// TIA Portal V20 export
FUNCTION_BLOCK "Sequence_1_ManualInput"   // FB126, LAD
TITLE = Sequence
// Sequence template programmend in ladder logic
// stored: IsIECCheckEnabled true, MemoryReserve 100, Namespace Unit1.Em5, SetENOAutomatically true
   VAR
      statSelectedJobNumber { ExternalWritable := 'False'} : DInt;   // Evaluated Job Number
      instSequenceLADControl { ExternalWritable := 'False'} : "LAF_ControlLadSequence";
      instSequenceLADStatus { ExternalWritable := 'False'} : "LAF_StatusLadSequence";
      statAxisCmdNumber { ExternalWritable := 'False'} : Array[0..1] of USInt;
      statTwoWayActCmdNumber { ExternalWritable := 'False'} : Array[0..3] of USInt;
      statPulse { ExternalWritable := 'False'} : Array[0..999] of Bool;
      statTonTimer { ExternalWritable := 'False'} : Array[0..999] of TON_TIME;
   END_VAR
   VAR_TEMP
      tempCustomerAction : Bool;   // Placeholder for possible actions
      tempDo_nothing_and_wait_for_init : Bool;   // Placeholder for doing nothing
      tempSafeStateCondition : Bool;   // Temp Condition for the equipment module to be in a safe state
   END_VAR
   VAR CONSTANT
      STEP_IDLE : DInt := 1;   // Idle Step
      JOB_1_STEP_01 : DInt := 101;   // Template Step
      JOB_1_STEP_11 : DInt := 111;   // Template Step
      JOB_1_STEP_21 : DInt := 121;   // Template Step
      JOB_1_STEP_31 : DInt := 131;   // Template Step
      JOB_1_STEP_41 : DInt := 141;
      JOB_1_STEP_51 : DInt := 151;
      JOB_1_STEP_91 : DInt := 191;
      JOB_2_STEP_01 : DInt := 201;   // Template Step
      JOB_2_STEP_11 : DInt := 211;   // Template Step
      JOB_2_STEP_21 : DInt := 221;   // Template Step
      JOB_2_STEP_31 : DInt := 231;   // Template Step
      JOB_2_STEP_41 : DInt := 241;   // Template Step
      JOB_2_STEP_51 : DInt := 251;   // Template Step
      JOB_2_STEP_61 : DInt := 261;   // Template Step
      JOB_2_STEP_91 : DInt := 291;   // Template Step
      JOB_3_STEP_01 : DInt := 301;   // Template Step
      JOB_3_STEP_11 : DInt := 311;   // Template Step
      JOB_3_STEP_21 : DInt := 321;   // Template Step
      JOB_3_STEP_31 : DInt := 331;   // Template Step
      JOB_3_STEP_41 : DInt := 341;   // Template Step
      JOB_3_STEP_51 : DInt := 351;   // Template Step
      JOB_3_STEP_91 : DInt := 391;   // Template Step
      STEP_IMMEDIATE_STOP : DInt := 901;   // Step executed when an immediate stop command is triggered for the sequence (i.e. when unit is in state aborting)
      SeqDelayTime : Time := T#100ms;
      SeqNoDelayTime : Time := T#0ms;
      TRUE : Bool := TRUE;
      FALSE : Bool := FALSE;
      NgAndManualInputAxisYHomePos : SInt := 0;
      NgAndManualInputAxisYWorkPos : SInt := 1;
   END_VAR
   // // statAxisCmdNumber[0] : cmNgAndManualInputAxisY
   // // statAxisCmdNumber[1] : cmMagazineAxisZ
   // // statTwoWayActCmdNumber[0] : cmNgAndManualInputCylinderUpDown
   // // statTwoWayActCmdNumber[1] : cmNgAndManualInputVacuum1OnOff
   // // statTwoWayActCmdNumber[2] : cmNgAndManualInputVacuum2OnOff
   // // statTwoWayActCmdNumber[3] : cmMagazineLockCylinderUpDown
   VAR_TEMP   // added for the SCL form of the ladder/FBD networks
      _w1 : Bool;
      _w2 : Bool;
      _w3 : Bool;
   END_VAR
BEGIN

REGION Network 1: BLOCK INFO HEADER
   // (company) / (C) Copyright (year)
   // ---------------------------------------------------------------------------------
   // Title:                             (Title of this block)
   // Comment/Function: (that is implemented in the block)
   // Library/Family:           (that the source is dedicated to)
   // Author:                        (department / person in charge / contact)
   // Target System:          (test system with FW version)
   // Engineering:              TIA Portal (SW version)
   // Restrictions:               (OB types, etc.)
   // Requirements:           (hardware, technological package, etc.)
   // ---------------------------------------------------------------------------------
   // Change log table:
   // Version          | Date             | Signature      | Expert in charge  | Changes applied ------------------------|----------------------|-------------------------|--------------------------------|-----------------------
   // 001.000.000 | yyyy-mm-dd | 0x00000000 | (name of expert) | First released version
END_REGION

REGION Network 2: DESCRIPTION
   // This is a template block provided by the Automation Framework. It can be used to create an own project.
   // The Block Info Header is prepared to put in your own data.
   // Description of the block could be added here and the docu created by Code2Docu.
END_REGION

REGION Network 3: ******************** CONTROL ********************
END_REGION

REGION Network 4: Sequence Control
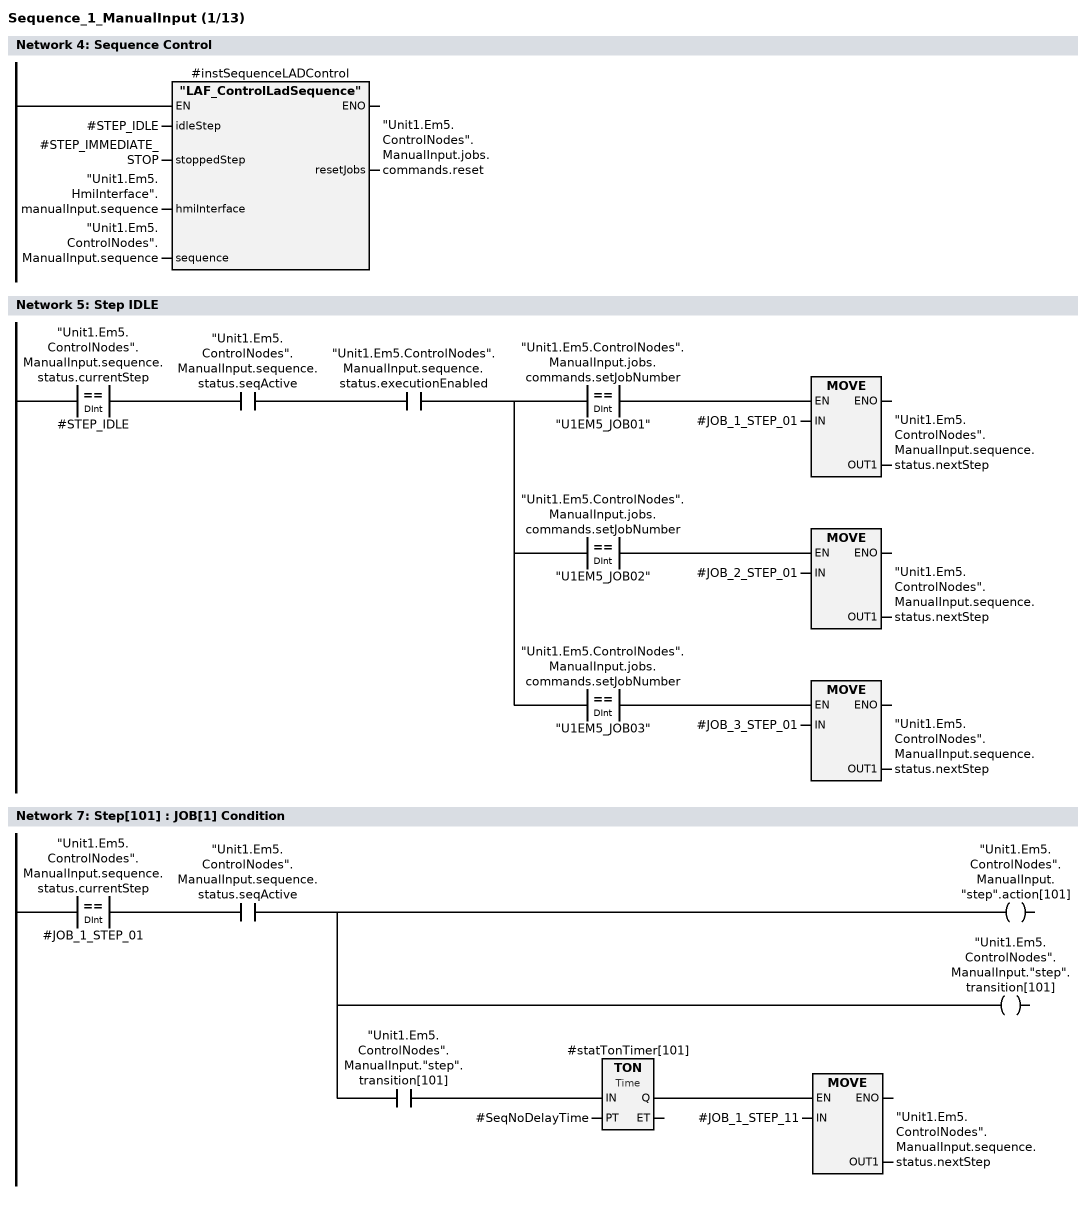
   RUNG wire#powerrail
      #instSequenceLADControl(idleStep := #STEP_IDLE, stoppedStep := #STEP_IMMEDIATE_STOP, hmiInterface := "Unit1.Em5.HmiInterface".manualInput.sequence, sequence := "Unit1.Em5.ControlNodes".ManualInput.sequence, resetJobs => "Unit1.Em5.ControlNodes".ManualInput.jobs.commands.reset)
   END_RUNG
   // the same network as SCL:
   #instSequenceLADControl(idleStep := #STEP_IDLE,   // "LAF_ControlLadSequence"
                           stoppedStep := #STEP_IMMEDIATE_STOP,
                           hmiInterface := "Unit1.Em5.HmiInterface".manualInput.sequence,
                           sequence := "Unit1.Em5.ControlNodes".ManualInput.sequence,
                           resetJobs => "Unit1.Em5.ControlNodes".ManualInput.jobs.commands.reset);
END_REGION

REGION Network 5: Step IDLE
   RUNG wire#powerrail
      { S7_Templates := "SrcType := DInt" } EQ_Contact(in1 := "Unit1.Em5.ControlNodes".ManualInput.sequence.status.currentStep, in2 := #STEP_IDLE)
      Contact( "Unit1.Em5.ControlNodes".ManualInput.sequence.status.seqActive )
      Contact( "Unit1.Em5.ControlNodes".ManualInput.sequence.status.executionEnabled )
      wire#w1
      { S7_Templates := "SrcType := DInt" } EQ_Contact(in1 := "Unit1.Em5.ControlNodes".ManualInput.jobs.commands.setJobNumber, in2 := "U1EM5_JOB01")
      Move(in := #JOB_1_STEP_01, out1 => "Unit1.Em5.ControlNodes".ManualInput.sequence.status.nextStep)
   END_RUNG
   RUNG wire#w1
      { S7_Templates := "SrcType := DInt" } EQ_Contact(in1 := "Unit1.Em5.ControlNodes".ManualInput.jobs.commands.setJobNumber, in2 := "U1EM5_JOB02")
      Move(in := #JOB_2_STEP_01, out1 => "Unit1.Em5.ControlNodes".ManualInput.sequence.status.nextStep)
   END_RUNG
   RUNG wire#w1
      { S7_Templates := "SrcType := DInt" } EQ_Contact(in1 := "Unit1.Em5.ControlNodes".ManualInput.jobs.commands.setJobNumber, in2 := "U1EM5_JOB03")
      Move(in := #JOB_3_STEP_01, out1 => "Unit1.Em5.ControlNodes".ManualInput.sequence.status.nextStep)
   END_RUNG
   // the same network as SCL:
   #_w1 := ("Unit1.Em5.ControlNodes".ManualInput.sequence.status.currentStep = #STEP_IDLE) AND "Unit1.Em5.ControlNodes".ManualInput.sequence.status.seqActive AND "Unit1.Em5.ControlNodes".ManualInput.sequence.status.executionEnabled;
   IF #_w1 AND ("Unit1.Em5.ControlNodes".ManualInput.jobs.commands.setJobNumber = "U1EM5_JOB01") THEN
       "Unit1.Em5.ControlNodes".ManualInput.sequence.status.nextStep := #JOB_1_STEP_01;
   END_IF;
   IF #_w1 AND ("Unit1.Em5.ControlNodes".ManualInput.jobs.commands.setJobNumber = "U1EM5_JOB02") THEN
       "Unit1.Em5.ControlNodes".ManualInput.sequence.status.nextStep := #JOB_2_STEP_01;
   END_IF;
   IF #_w1 AND ("Unit1.Em5.ControlNodes".ManualInput.jobs.commands.setJobNumber = "U1EM5_JOB03") THEN
       "Unit1.Em5.ControlNodes".ManualInput.sequence.status.nextStep := #JOB_3_STEP_01;
   END_IF;
END_REGION

REGION Network 6: ******************** JOB[1] EM INITIALIZED ********************
END_REGION

REGION Network 7: Step[101] : JOB[1] Condition
   RUNG wire#powerrail
      { S7_Templates := "SrcType := DInt" } EQ_Contact(in1 := "Unit1.Em5.ControlNodes".ManualInput.sequence.status.currentStep, in2 := #JOB_1_STEP_01)
      Contact( "Unit1.Em5.ControlNodes".ManualInput.sequence.status.seqActive )
      wire#w1
      Coil( "Unit1.Em5.ControlNodes".ManualInput."step".action[101] )
   END_RUNG
   RUNG wire#w1
      Coil( "Unit1.Em5.ControlNodes".ManualInput."step".transition[101] )
   END_RUNG
   RUNG wire#w1
      Contact( "Unit1.Em5.ControlNodes".ManualInput."step".transition[101] )
      { S7_Templates := "time_type := Time" } #statTonTimer[101].TON(pt := #SeqNoDelayTime, et =>)
      Move(in := #JOB_1_STEP_11, out1 => "Unit1.Em5.ControlNodes".ManualInput.sequence.status.nextStep)
   END_RUNG
   // the same network as SCL:
   "Unit1.Em5.ControlNodes".ManualInput."step".action[101] := ("Unit1.Em5.ControlNodes".ManualInput.sequence.status.currentStep = #JOB_1_STEP_01) AND "Unit1.Em5.ControlNodes".ManualInput.sequence.status.seqActive;
   "Unit1.Em5.ControlNodes".ManualInput."step".transition[101] := ("Unit1.Em5.ControlNodes".ManualInput.sequence.status.currentStep = #JOB_1_STEP_01) AND "Unit1.Em5.ControlNodes".ManualInput.sequence.status.seqActive;
   #statTonTimer[101].TON(IN := ("Unit1.Em5.ControlNodes".ManualInput.sequence.status.currentStep = #JOB_1_STEP_01) AND "Unit1.Em5.ControlNodes".ManualInput.sequence.status.seqActive AND "Unit1.Em5.ControlNodes".ManualInput."step".transition[101],
                          PT := #SeqNoDelayTime);
   IF #statTonTimer[101].Q THEN
       "Unit1.Em5.ControlNodes".ManualInput.sequence.status.nextStep := #JOB_1_STEP_11;
   END_IF;
END_REGION

REGION Network 8: Step[111] : Ng And Manual Input Cylinder HomePos & Magazine Lock Cylinder WorkPos Check
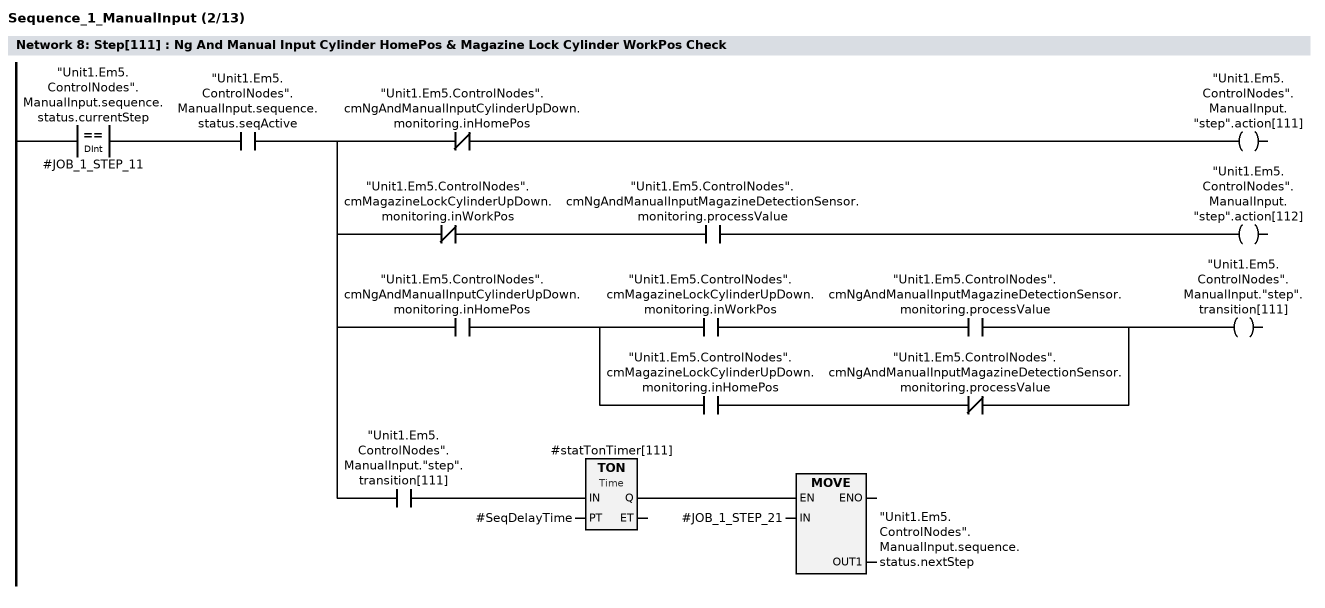
   RUNG wire#powerrail
      { S7_Templates := "SrcType := DInt" } EQ_Contact(in1 := "Unit1.Em5.ControlNodes".ManualInput.sequence.status.currentStep, in2 := #JOB_1_STEP_11)
      Contact( "Unit1.Em5.ControlNodes".ManualInput.sequence.status.seqActive )
      wire#w1
      I_Contact( "Unit1.Em5.ControlNodes".cmNgAndManualInputCylinderUpDown.monitoring.inHomePos )
      Coil( "Unit1.Em5.ControlNodes".ManualInput."step".action[111] )
   END_RUNG
   RUNG wire#w1
      I_Contact( "Unit1.Em5.ControlNodes".cmMagazineLockCylinderUpDown.monitoring.inWorkPos )
      Contact( "Unit1.Em5.ControlNodes".cmNgAndManualInputMagazineDetectionSensor.monitoring.processValue )
      Coil( "Unit1.Em5.ControlNodes".ManualInput."step".action[112] )
   END_RUNG
   RUNG wire#w1
      Contact( "Unit1.Em5.ControlNodes".cmNgAndManualInputCylinderUpDown.monitoring.inHomePos )
      wire#w2
      Contact( "Unit1.Em5.ControlNodes".cmMagazineLockCylinderUpDown.monitoring.inWorkPos )
      Contact( "Unit1.Em5.ControlNodes".cmNgAndManualInputMagazineDetectionSensor.monitoring.processValue )
      wire#w3
      Coil( "Unit1.Em5.ControlNodes".ManualInput."step".transition[111] )
   END_RUNG
   RUNG wire#w2
      Contact( "Unit1.Em5.ControlNodes".cmMagazineLockCylinderUpDown.monitoring.inHomePos )
      I_Contact( "Unit1.Em5.ControlNodes".cmNgAndManualInputMagazineDetectionSensor.monitoring.processValue )
   END_RUNG wire#w3
   RUNG wire#w1
      Contact( "Unit1.Em5.ControlNodes".ManualInput."step".transition[111] )
      { S7_Templates := "time_type := Time" } #statTonTimer[111].TON(pt := #SeqDelayTime, et =>)
      Move(in := #JOB_1_STEP_21, out1 => "Unit1.Em5.ControlNodes".ManualInput.sequence.status.nextStep)
   END_RUNG
   // the same network as SCL:
   #_w1 := ("Unit1.Em5.ControlNodes".ManualInput.sequence.status.currentStep = #JOB_1_STEP_11) AND "Unit1.Em5.ControlNodes".ManualInput.sequence.status.seqActive;
   "Unit1.Em5.ControlNodes".ManualInput."step".action[111] := #_w1 AND NOT "Unit1.Em5.ControlNodes".cmNgAndManualInputCylinderUpDown.monitoring.inHomePos;
   "Unit1.Em5.ControlNodes".ManualInput."step".action[112] := #_w1 AND NOT "Unit1.Em5.ControlNodes".cmMagazineLockCylinderUpDown.monitoring.inWorkPos AND "Unit1.Em5.ControlNodes".cmNgAndManualInputMagazineDetectionSensor.monitoring.processValue;
   "Unit1.Em5.ControlNodes".ManualInput."step".transition[111] := #_w1 AND "Unit1.Em5.ControlNodes".cmNgAndManualInputCylinderUpDown.monitoring.inHomePos AND (("Unit1.Em5.ControlNodes".cmMagazineLockCylinderUpDown.monitoring.inWorkPos AND "Unit1.Em5.ControlNodes".cmNgAndManualInputMagazineDetectionSensor.monitoring.processValue) OR ("Unit1.Em5.ControlNodes".cmMagazineLockCylinderUpDown.monitoring.inHomePos AND NOT "Unit1.Em5.ControlNodes".cmNgAndManualInputMagazineDetectionSensor.monitoring.processValue));
   #statTonTimer[111].TON(IN := #_w1 AND "Unit1.Em5.ControlNodes".ManualInput."step".transition[111],
                          PT := #SeqDelayTime);
   IF #statTonTimer[111].Q THEN
       "Unit1.Em5.ControlNodes".ManualInput.sequence.status.nextStep := #JOB_1_STEP_21;
   END_IF;
END_REGION

REGION Network 9: Step[121] : Ng And Manual Input Vacuum HomePos & Vibrator Home Pos Check
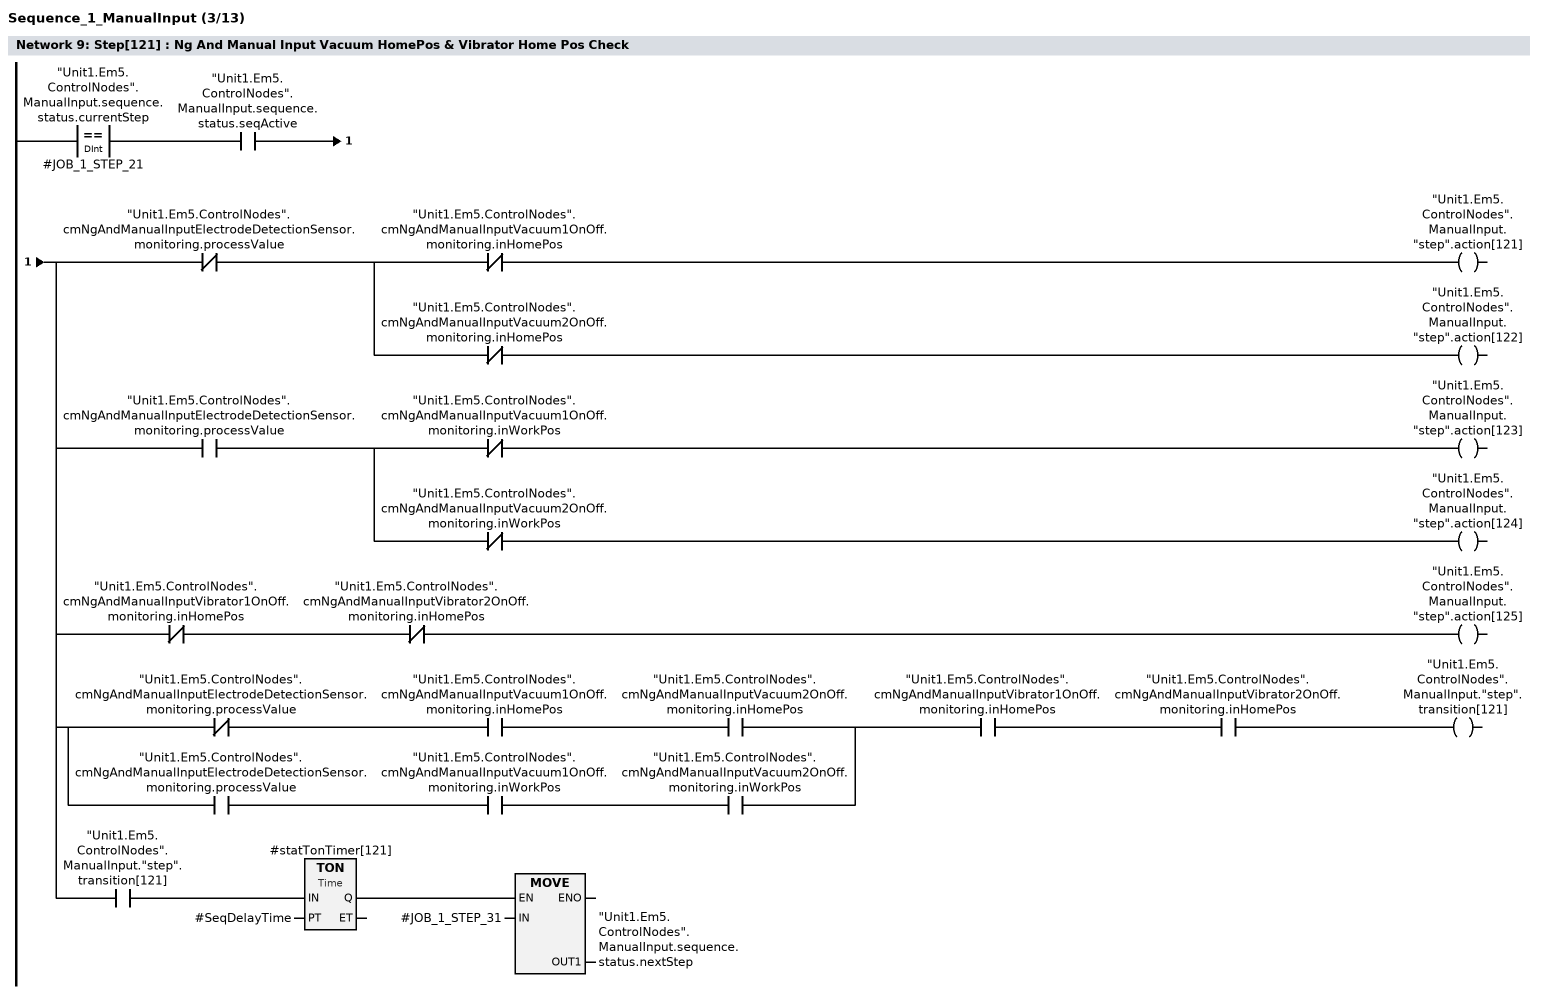
   RUNG wire#powerrail
      { S7_Templates := "SrcType := DInt" } EQ_Contact(in1 := "Unit1.Em5.ControlNodes".ManualInput.sequence.status.currentStep, in2 := #JOB_1_STEP_21)
      Contact( "Unit1.Em5.ControlNodes".ManualInput.sequence.status.seqActive )
      wire#w1
      I_Contact( "Unit1.Em5.ControlNodes".cmNgAndManualInputElectrodeDetectionSensor.monitoring.processValue )
      wire#w2
      I_Contact( "Unit1.Em5.ControlNodes".cmNgAndManualInputVacuum1OnOff.monitoring.inHomePos )
      Coil( "Unit1.Em5.ControlNodes".ManualInput."step".action[121] )
   END_RUNG
   RUNG wire#w2
      I_Contact( "Unit1.Em5.ControlNodes".cmNgAndManualInputVacuum2OnOff.monitoring.inHomePos )
      Coil( "Unit1.Em5.ControlNodes".ManualInput."step".action[122] )
   END_RUNG
   RUNG wire#w1
      Contact( "Unit1.Em5.ControlNodes".cmNgAndManualInputElectrodeDetectionSensor.monitoring.processValue )
      wire#w3
      I_Contact( "Unit1.Em5.ControlNodes".cmNgAndManualInputVacuum1OnOff.monitoring.inWorkPos )
      Coil( "Unit1.Em5.ControlNodes".ManualInput."step".action[123] )
   END_RUNG
   RUNG wire#w3
      I_Contact( "Unit1.Em5.ControlNodes".cmNgAndManualInputVacuum2OnOff.monitoring.inWorkPos )
      Coil( "Unit1.Em5.ControlNodes".ManualInput."step".action[124] )
   END_RUNG
   RUNG wire#w1
      I_Contact( "Unit1.Em5.ControlNodes".cmNgAndManualInputVibrator1OnOff.monitoring.inHomePos )
      I_Contact( "Unit1.Em5.ControlNodes".cmNgAndManualInputVibrator2OnOff.monitoring.inHomePos )
      Coil( "Unit1.Em5.ControlNodes".ManualInput."step".action[125] )
   END_RUNG
   RUNG wire#w1
      I_Contact( "Unit1.Em5.ControlNodes".cmNgAndManualInputElectrodeDetectionSensor.monitoring.processValue )
      Contact( "Unit1.Em5.ControlNodes".cmNgAndManualInputVacuum1OnOff.monitoring.inHomePos )
      Contact( "Unit1.Em5.ControlNodes".cmNgAndManualInputVacuum2OnOff.monitoring.inHomePos )
      wire#w4
      Contact( "Unit1.Em5.ControlNodes".cmNgAndManualInputVibrator1OnOff.monitoring.inHomePos )
      Contact( "Unit1.Em5.ControlNodes".cmNgAndManualInputVibrator2OnOff.monitoring.inHomePos )
      Coil( "Unit1.Em5.ControlNodes".ManualInput."step".transition[121] )
   END_RUNG
   RUNG wire#w1
      Contact( "Unit1.Em5.ControlNodes".cmNgAndManualInputElectrodeDetectionSensor.monitoring.processValue )
      Contact( "Unit1.Em5.ControlNodes".cmNgAndManualInputVacuum1OnOff.monitoring.inWorkPos )
      Contact( "Unit1.Em5.ControlNodes".cmNgAndManualInputVacuum2OnOff.monitoring.inWorkPos )
   END_RUNG wire#w4
   RUNG wire#w1
      Contact( "Unit1.Em5.ControlNodes".ManualInput."step".transition[121] )
      { S7_Templates := "time_type := Time" } #statTonTimer[121].TON(pt := #SeqDelayTime, et =>)
      Move(in := #JOB_1_STEP_31, out1 => "Unit1.Em5.ControlNodes".ManualInput.sequence.status.nextStep)
   END_RUNG
   // the same network as SCL:
   #_w1 := ("Unit1.Em5.ControlNodes".ManualInput.sequence.status.currentStep = #JOB_1_STEP_21) AND "Unit1.Em5.ControlNodes".ManualInput.sequence.status.seqActive;
   #_w2 := #_w1 AND NOT "Unit1.Em5.ControlNodes".cmNgAndManualInputElectrodeDetectionSensor.monitoring.processValue;
   "Unit1.Em5.ControlNodes".ManualInput."step".action[121] := #_w2 AND NOT "Unit1.Em5.ControlNodes".cmNgAndManualInputVacuum1OnOff.monitoring.inHomePos;
   "Unit1.Em5.ControlNodes".ManualInput."step".action[122] := #_w2 AND NOT "Unit1.Em5.ControlNodes".cmNgAndManualInputVacuum2OnOff.monitoring.inHomePos;
   #_w3 := #_w1 AND "Unit1.Em5.ControlNodes".cmNgAndManualInputElectrodeDetectionSensor.monitoring.processValue;
   "Unit1.Em5.ControlNodes".ManualInput."step".action[123] := #_w3 AND NOT "Unit1.Em5.ControlNodes".cmNgAndManualInputVacuum1OnOff.monitoring.inWorkPos;
   "Unit1.Em5.ControlNodes".ManualInput."step".action[124] := #_w3 AND NOT "Unit1.Em5.ControlNodes".cmNgAndManualInputVacuum2OnOff.monitoring.inWorkPos;
   "Unit1.Em5.ControlNodes".ManualInput."step".action[125] := #_w1 AND NOT "Unit1.Em5.ControlNodes".cmNgAndManualInputVibrator1OnOff.monitoring.inHomePos AND NOT "Unit1.Em5.ControlNodes".cmNgAndManualInputVibrator2OnOff.monitoring.inHomePos;
   "Unit1.Em5.ControlNodes".ManualInput."step".transition[121] := #_w1 AND ((NOT "Unit1.Em5.ControlNodes".cmNgAndManualInputElectrodeDetectionSensor.monitoring.processValue AND "Unit1.Em5.ControlNodes".cmNgAndManualInputVacuum1OnOff.monitoring.inHomePos AND "Unit1.Em5.ControlNodes".cmNgAndManualInputVacuum2OnOff.monitoring.inHomePos) OR ("Unit1.Em5.ControlNodes".cmNgAndManualInputElectrodeDetectionSensor.monitoring.processValue AND "Unit1.Em5.ControlNodes".cmNgAndManualInputVacuum1OnOff.monitoring.inWorkPos AND "Unit1.Em5.ControlNodes".cmNgAndManualInputVacuum2OnOff.monitoring.inWorkPos)) AND "Unit1.Em5.ControlNodes".cmNgAndManualInputVibrator1OnOff.monitoring.inHomePos AND "Unit1.Em5.ControlNodes".cmNgAndManualInputVibrator2OnOff.monitoring.inHomePos;
   #statTonTimer[121].TON(IN := #_w1 AND "Unit1.Em5.ControlNodes".ManualInput."step".transition[121],
                          PT := #SeqDelayTime);
   IF #statTonTimer[121].Q THEN
       "Unit1.Em5.ControlNodes".ManualInput.sequence.status.nextStep := #JOB_1_STEP_31;
   END_IF;
END_REGION

REGION Network 10: Step[131] : Ng And Manual Input AxisY & Magazine AxisZ Homed Check
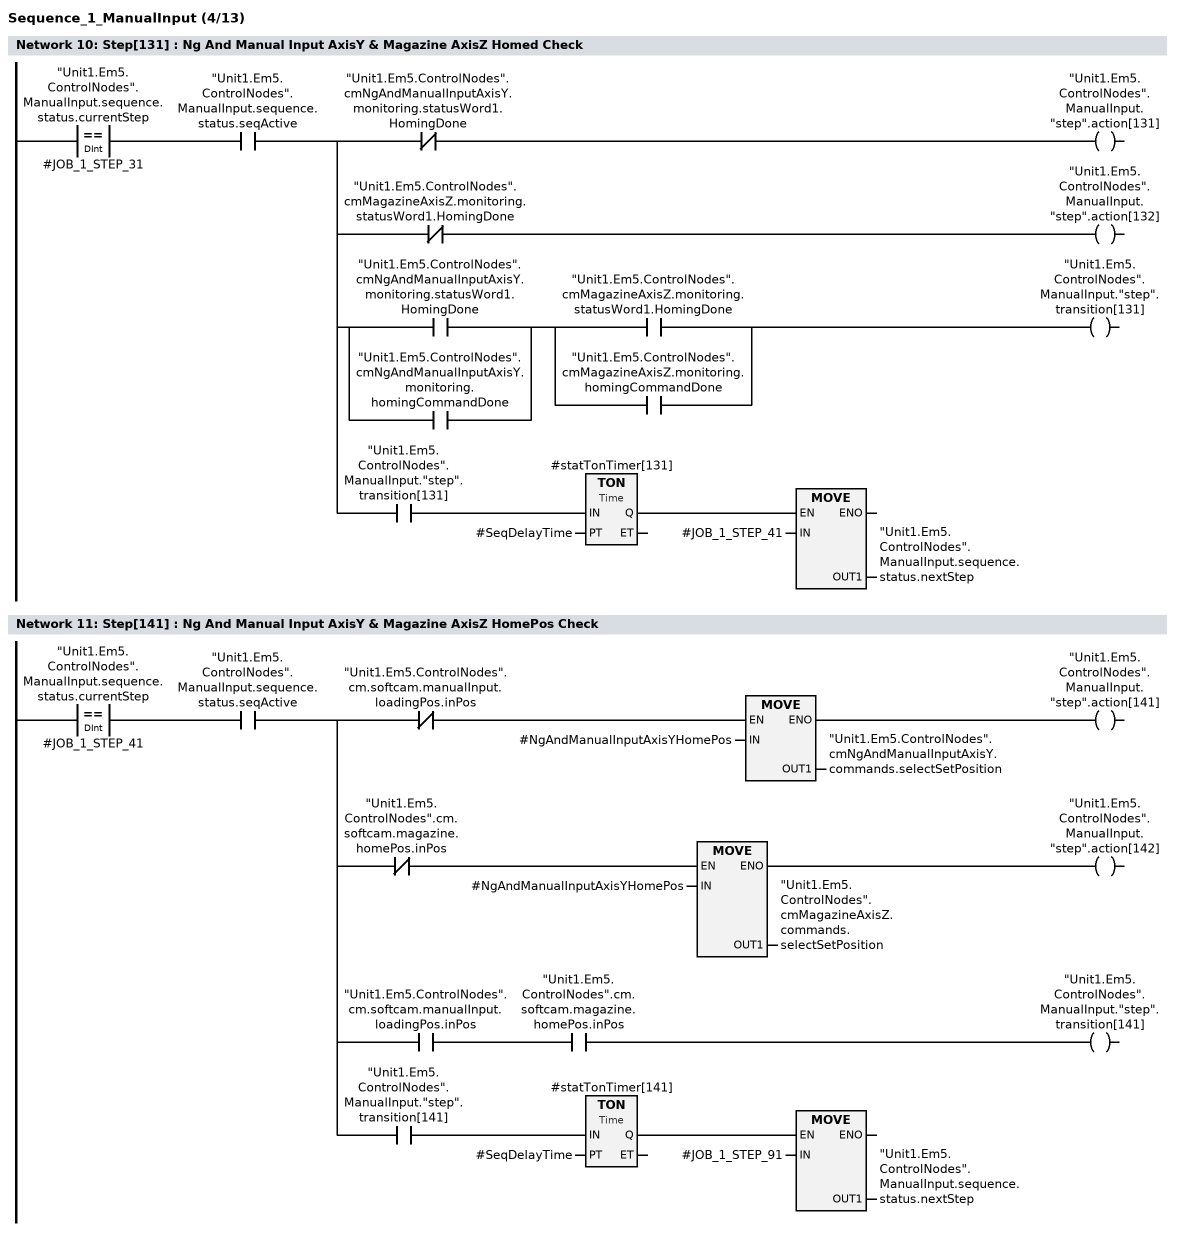
   RUNG wire#powerrail
      { S7_Templates := "SrcType := DInt" } EQ_Contact(in1 := "Unit1.Em5.ControlNodes".ManualInput.sequence.status.currentStep, in2 := #JOB_1_STEP_31)
      Contact( "Unit1.Em5.ControlNodes".ManualInput.sequence.status.seqActive )
      wire#w1
      I_Contact( "Unit1.Em5.ControlNodes".cmNgAndManualInputAxisY.monitoring.statusWord1.HomingDone )
      Coil( "Unit1.Em5.ControlNodes".ManualInput."step".action[131] )
   END_RUNG
   RUNG wire#w1
      I_Contact( "Unit1.Em5.ControlNodes".cmMagazineAxisZ.monitoring.statusWord1.HomingDone )
      Coil( "Unit1.Em5.ControlNodes".ManualInput."step".action[132] )
   END_RUNG
   RUNG wire#w1
      Contact( "Unit1.Em5.ControlNodes".cmNgAndManualInputAxisY.monitoring.statusWord1.HomingDone )
      wire#w2
      Contact( "Unit1.Em5.ControlNodes".cmMagazineAxisZ.monitoring.statusWord1.HomingDone )
      wire#w3
      Coil( "Unit1.Em5.ControlNodes".ManualInput."step".transition[131] )
   END_RUNG
   RUNG wire#w1
      Contact( "Unit1.Em5.ControlNodes".cmNgAndManualInputAxisY.monitoring.homingCommandDone )
   END_RUNG wire#w2
   RUNG wire#w2
      Contact( "Unit1.Em5.ControlNodes".cmMagazineAxisZ.monitoring.homingCommandDone )
   END_RUNG wire#w3
   RUNG wire#w1
      Contact( "Unit1.Em5.ControlNodes".ManualInput."step".transition[131] )
      { S7_Templates := "time_type := Time" } #statTonTimer[131].TON(pt := #SeqDelayTime, et =>)
      Move(in := #JOB_1_STEP_41, out1 => "Unit1.Em5.ControlNodes".ManualInput.sequence.status.nextStep)
   END_RUNG
   // the same network as SCL:
   #_w1 := ("Unit1.Em5.ControlNodes".ManualInput.sequence.status.currentStep = #JOB_1_STEP_31) AND "Unit1.Em5.ControlNodes".ManualInput.sequence.status.seqActive;
   "Unit1.Em5.ControlNodes".ManualInput."step".action[131] := #_w1 AND NOT "Unit1.Em5.ControlNodes".cmNgAndManualInputAxisY.monitoring.statusWord1.HomingDone;
   "Unit1.Em5.ControlNodes".ManualInput."step".action[132] := #_w1 AND NOT "Unit1.Em5.ControlNodes".cmMagazineAxisZ.monitoring.statusWord1.HomingDone;
   "Unit1.Em5.ControlNodes".ManualInput."step".transition[131] := #_w1 AND ("Unit1.Em5.ControlNodes".cmNgAndManualInputAxisY.monitoring.statusWord1.HomingDone OR "Unit1.Em5.ControlNodes".cmNgAndManualInputAxisY.monitoring.homingCommandDone) AND ("Unit1.Em5.ControlNodes".cmMagazineAxisZ.monitoring.statusWord1.HomingDone OR "Unit1.Em5.ControlNodes".cmMagazineAxisZ.monitoring.homingCommandDone);
   #statTonTimer[131].TON(IN := #_w1 AND "Unit1.Em5.ControlNodes".ManualInput."step".transition[131],
                          PT := #SeqDelayTime);
   IF #statTonTimer[131].Q THEN
       "Unit1.Em5.ControlNodes".ManualInput.sequence.status.nextStep := #JOB_1_STEP_41;
   END_IF;
END_REGION

REGION Network 11: Step[141] : Ng And Manual Input AxisY & Magazine AxisZ HomePos Check
   RUNG wire#powerrail
      { S7_Templates := "SrcType := DInt" } EQ_Contact(in1 := "Unit1.Em5.ControlNodes".ManualInput.sequence.status.currentStep, in2 := #JOB_1_STEP_41)
      Contact( "Unit1.Em5.ControlNodes".ManualInput.sequence.status.seqActive )
      wire#w1
      I_Contact( "Unit1.Em5.ControlNodes".cm.softcam.manualInput.loadingPos.inPos )
      Move(in := #NgAndManualInputAxisYHomePos, out1 => "Unit1.Em5.ControlNodes".cmNgAndManualInputAxisY.commands.selectSetPosition)
      Coil( "Unit1.Em5.ControlNodes".ManualInput."step".action[141] )
   END_RUNG
   RUNG wire#w1
      I_Contact( "Unit1.Em5.ControlNodes".cm.softcam.magazine.homePos.inPos )
      Move(in := #NgAndManualInputAxisYHomePos, out1 => "Unit1.Em5.ControlNodes".cmMagazineAxisZ.commands.selectSetPosition)
      Coil( "Unit1.Em5.ControlNodes".ManualInput."step".action[142] )
   END_RUNG
   RUNG wire#w1
      Contact( "Unit1.Em5.ControlNodes".cm.softcam.manualInput.loadingPos.inPos )
      Contact( "Unit1.Em5.ControlNodes".cm.softcam.magazine.homePos.inPos )
      Coil( "Unit1.Em5.ControlNodes".ManualInput."step".transition[141] )
   END_RUNG
   RUNG wire#w1
      Contact( "Unit1.Em5.ControlNodes".ManualInput."step".transition[141] )
      { S7_Templates := "time_type := Time" } #statTonTimer[141].TON(pt := #SeqDelayTime, et =>)
      Move(in := #JOB_1_STEP_91, out1 => "Unit1.Em5.ControlNodes".ManualInput.sequence.status.nextStep)
   END_RUNG
   // the same network as SCL:
   #_w1 := ("Unit1.Em5.ControlNodes".ManualInput.sequence.status.currentStep = #JOB_1_STEP_41) AND "Unit1.Em5.ControlNodes".ManualInput.sequence.status.seqActive;
   #_w2 := #_w1 AND NOT "Unit1.Em5.ControlNodes".cm.softcam.manualInput.loadingPos.inPos;
   IF #_w2 THEN
       "Unit1.Em5.ControlNodes".cmNgAndManualInputAxisY.commands.selectSetPosition := #NgAndManualInputAxisYHomePos;
   END_IF;
   "Unit1.Em5.ControlNodes".ManualInput."step".action[141] := #_w2;
   #_w3 := #_w1 AND NOT "Unit1.Em5.ControlNodes".cm.softcam.magazine.homePos.inPos;
   IF #_w3 THEN
       "Unit1.Em5.ControlNodes".cmMagazineAxisZ.commands.selectSetPosition := #NgAndManualInputAxisYHomePos;
   END_IF;
   "Unit1.Em5.ControlNodes".ManualInput."step".action[142] := #_w3;
   "Unit1.Em5.ControlNodes".ManualInput."step".transition[141] := #_w1 AND "Unit1.Em5.ControlNodes".cm.softcam.manualInput.loadingPos.inPos AND "Unit1.Em5.ControlNodes".cm.softcam.magazine.homePos.inPos;
   #statTonTimer[141].TON(IN := #_w1 AND "Unit1.Em5.ControlNodes".ManualInput."step".transition[141],
                          PT := #SeqDelayTime);
   IF #statTonTimer[141].Q THEN
       "Unit1.Em5.ControlNodes".ManualInput.sequence.status.nextStep := #JOB_1_STEP_91;
   END_IF;
END_REGION

REGION Network 12: Step[151] : Magazine AxisZ PickUpPos Check
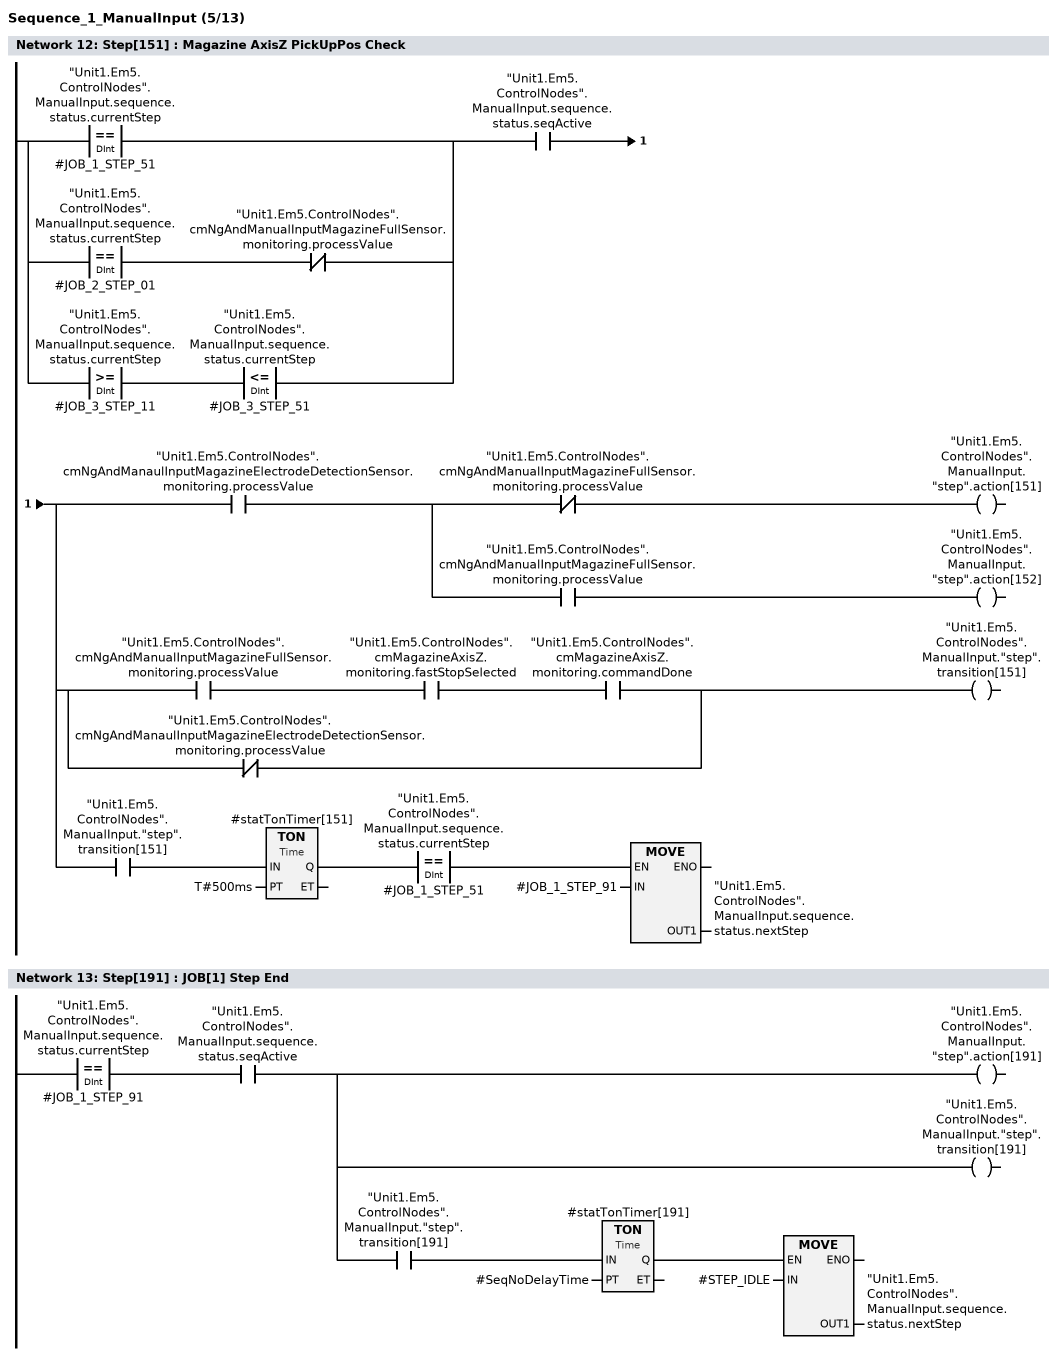
   RUNG wire#powerrail
      { S7_Templates := "SrcType := DInt" } EQ_Contact(in1 := "Unit1.Em5.ControlNodes".ManualInput.sequence.status.currentStep, in2 := #JOB_1_STEP_51)
      wire#w1
      Contact( "Unit1.Em5.ControlNodes".ManualInput.sequence.status.seqActive )
      wire#w2
      Contact( "Unit1.Em5.ControlNodes".cmNgAndManaulInputMagazineElectrodeDetectionSensor.monitoring.processValue )
      wire#w3
      I_Contact( "Unit1.Em5.ControlNodes".cmNgAndManualInputMagazineFullSensor.monitoring.processValue )
      Coil( "Unit1.Em5.ControlNodes".ManualInput."step".action[151] )
   END_RUNG
   RUNG wire#powerrail
      { S7_Templates := "SrcType := DInt" } EQ_Contact(in1 := "Unit1.Em5.ControlNodes".ManualInput.sequence.status.currentStep, in2 := #JOB_2_STEP_01)
      I_Contact( "Unit1.Em5.ControlNodes".cmNgAndManualInputMagazineFullSensor.monitoring.processValue )
   END_RUNG wire#w1
   RUNG wire#powerrail
      { S7_Templates := "SrcType := DInt" } GE_Contact(in1 := "Unit1.Em5.ControlNodes".ManualInput.sequence.status.currentStep, in2 := #JOB_3_STEP_11)
      { S7_Templates := "SrcType := DInt" } LE_Contact(in1 := "Unit1.Em5.ControlNodes".ManualInput.sequence.status.currentStep, in2 := #JOB_3_STEP_51)
   END_RUNG wire#w1
   RUNG wire#w3
      Contact( "Unit1.Em5.ControlNodes".cmNgAndManualInputMagazineFullSensor.monitoring.processValue )
      Coil( "Unit1.Em5.ControlNodes".ManualInput."step".action[152] )
   END_RUNG
   RUNG wire#w2
      Contact( "Unit1.Em5.ControlNodes".cmNgAndManualInputMagazineFullSensor.monitoring.processValue )
      Contact( "Unit1.Em5.ControlNodes".cmMagazineAxisZ.monitoring.fastStopSelected )
      Contact( "Unit1.Em5.ControlNodes".cmMagazineAxisZ.monitoring.commandDone )
      wire#w4
      Coil( "Unit1.Em5.ControlNodes".ManualInput."step".transition[151] )
   END_RUNG
   RUNG wire#w2
      I_Contact( "Unit1.Em5.ControlNodes".cmNgAndManaulInputMagazineElectrodeDetectionSensor.monitoring.processValue )
   END_RUNG wire#w4
   RUNG wire#w2
      Contact( "Unit1.Em5.ControlNodes".ManualInput."step".transition[151] )
      { S7_Templates := "time_type := Time" } #statTonTimer[151].TON(pt := T#500ms, et =>)
      { S7_Templates := "SrcType := DInt" } EQ_Contact(in1 := "Unit1.Em5.ControlNodes".ManualInput.sequence.status.currentStep, in2 := #JOB_1_STEP_51)
      Move(in := #JOB_1_STEP_91, out1 => "Unit1.Em5.ControlNodes".ManualInput.sequence.status.nextStep)
   END_RUNG
   // the same network as SCL:
   #_w1 := (("Unit1.Em5.ControlNodes".ManualInput.sequence.status.currentStep = #JOB_1_STEP_51) OR (("Unit1.Em5.ControlNodes".ManualInput.sequence.status.currentStep = #JOB_2_STEP_01) AND NOT "Unit1.Em5.ControlNodes".cmNgAndManualInputMagazineFullSensor.monitoring.processValue) OR (("Unit1.Em5.ControlNodes".ManualInput.sequence.status.currentStep >= #JOB_3_STEP_11) AND ("Unit1.Em5.ControlNodes".ManualInput.sequence.status.currentStep <= #JOB_3_STEP_51))) AND "Unit1.Em5.ControlNodes".ManualInput.sequence.status.seqActive;
   #_w2 := #_w1 AND "Unit1.Em5.ControlNodes".cmNgAndManaulInputMagazineElectrodeDetectionSensor.monitoring.processValue;
   "Unit1.Em5.ControlNodes".ManualInput."step".action[151] := #_w2 AND NOT "Unit1.Em5.ControlNodes".cmNgAndManualInputMagazineFullSensor.monitoring.processValue;
   "Unit1.Em5.ControlNodes".ManualInput."step".action[152] := #_w2 AND "Unit1.Em5.ControlNodes".cmNgAndManualInputMagazineFullSensor.monitoring.processValue;
   "Unit1.Em5.ControlNodes".ManualInput."step".transition[151] := #_w1 AND (("Unit1.Em5.ControlNodes".cmNgAndManualInputMagazineFullSensor.monitoring.processValue AND "Unit1.Em5.ControlNodes".cmMagazineAxisZ.monitoring.fastStopSelected AND "Unit1.Em5.ControlNodes".cmMagazineAxisZ.monitoring.commandDone) OR NOT "Unit1.Em5.ControlNodes".cmNgAndManaulInputMagazineElectrodeDetectionSensor.monitoring.processValue);
   #statTonTimer[151].TON(IN := #_w1 AND "Unit1.Em5.ControlNodes".ManualInput."step".transition[151],
                          PT := T#500ms);
   IF #statTonTimer[151].Q AND ("Unit1.Em5.ControlNodes".ManualInput.sequence.status.currentStep = #JOB_1_STEP_51) THEN
       "Unit1.Em5.ControlNodes".ManualInput.sequence.status.nextStep := #JOB_1_STEP_91;
   END_IF;
END_REGION

REGION Network 13: Step[191] : JOB[1] Step End
   RUNG wire#powerrail
      { S7_Templates := "SrcType := DInt" } EQ_Contact(in1 := "Unit1.Em5.ControlNodes".ManualInput.sequence.status.currentStep, in2 := #JOB_1_STEP_91)
      Contact( "Unit1.Em5.ControlNodes".ManualInput.sequence.status.seqActive )
      wire#w1
      Coil( "Unit1.Em5.ControlNodes".ManualInput."step".action[191] )
   END_RUNG
   RUNG wire#w1
      Coil( "Unit1.Em5.ControlNodes".ManualInput."step".transition[191] )
   END_RUNG
   RUNG wire#w1
      Contact( "Unit1.Em5.ControlNodes".ManualInput."step".transition[191] )
      { S7_Templates := "time_type := Time" } #statTonTimer[191].TON(pt := #SeqNoDelayTime, et =>)
      Move(in := #STEP_IDLE, out1 => "Unit1.Em5.ControlNodes".ManualInput.sequence.status.nextStep)
   END_RUNG
   // the same network as SCL:
   "Unit1.Em5.ControlNodes".ManualInput."step".action[191] := ("Unit1.Em5.ControlNodes".ManualInput.sequence.status.currentStep = #JOB_1_STEP_91) AND "Unit1.Em5.ControlNodes".ManualInput.sequence.status.seqActive;
   "Unit1.Em5.ControlNodes".ManualInput."step".transition[191] := ("Unit1.Em5.ControlNodes".ManualInput.sequence.status.currentStep = #JOB_1_STEP_91) AND "Unit1.Em5.ControlNodes".ManualInput.sequence.status.seqActive;
   #statTonTimer[191].TON(IN := ("Unit1.Em5.ControlNodes".ManualInput.sequence.status.currentStep = #JOB_1_STEP_91) AND "Unit1.Em5.ControlNodes".ManualInput.sequence.status.seqActive AND "Unit1.Em5.ControlNodes".ManualInput."step".transition[191],
                          PT := #SeqNoDelayTime);
   IF #statTonTimer[191].Q THEN
       "Unit1.Em5.ControlNodes".ManualInput.sequence.status.nextStep := #STEP_IDLE;
   END_IF;
END_REGION

REGION Network 14: ******************** JOB[2] LOADING AUTO ********************
END_REGION

REGION Network 15: Step[201] : JOB[2] Condition
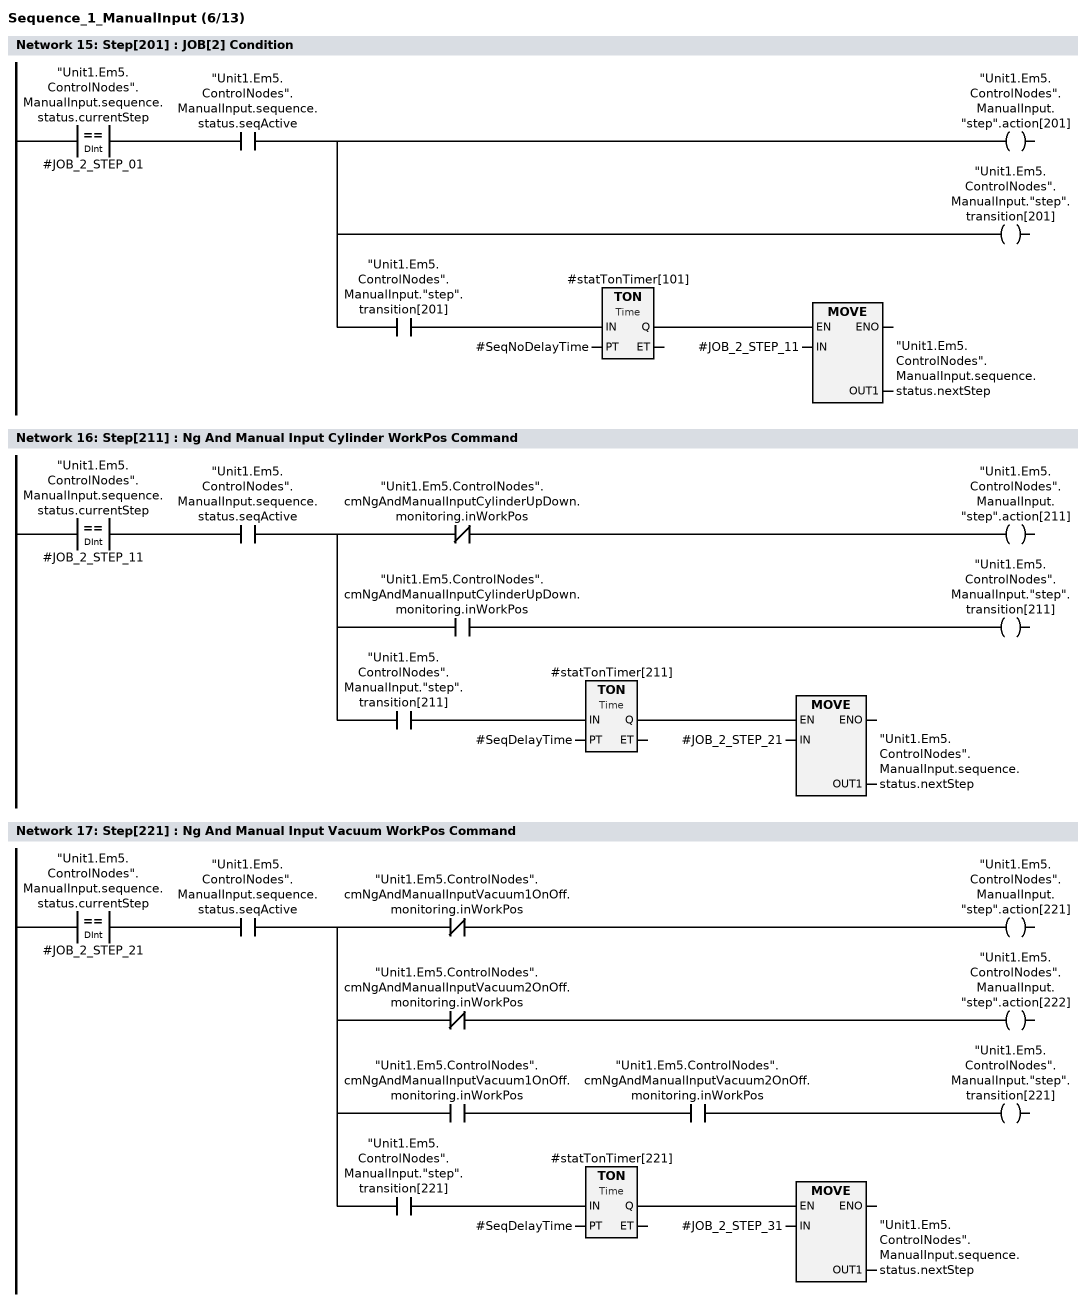
   RUNG wire#powerrail
      { S7_Templates := "SrcType := DInt" } EQ_Contact(in1 := "Unit1.Em5.ControlNodes".ManualInput.sequence.status.currentStep, in2 := #JOB_2_STEP_01)
      Contact( "Unit1.Em5.ControlNodes".ManualInput.sequence.status.seqActive )
      wire#w1
      Coil( "Unit1.Em5.ControlNodes".ManualInput."step".action[201] )
   END_RUNG
   RUNG wire#w1
      Coil( "Unit1.Em5.ControlNodes".ManualInput."step".transition[201] )
   END_RUNG
   RUNG wire#w1
      Contact( "Unit1.Em5.ControlNodes".ManualInput."step".transition[201] )
      { S7_Templates := "time_type := Time" } #statTonTimer[101].TON(pt := #SeqNoDelayTime, et =>)
      Move(in := #JOB_2_STEP_11, out1 => "Unit1.Em5.ControlNodes".ManualInput.sequence.status.nextStep)
   END_RUNG
   // the same network as SCL:
   "Unit1.Em5.ControlNodes".ManualInput."step".action[201] := ("Unit1.Em5.ControlNodes".ManualInput.sequence.status.currentStep = #JOB_2_STEP_01) AND "Unit1.Em5.ControlNodes".ManualInput.sequence.status.seqActive;
   "Unit1.Em5.ControlNodes".ManualInput."step".transition[201] := ("Unit1.Em5.ControlNodes".ManualInput.sequence.status.currentStep = #JOB_2_STEP_01) AND "Unit1.Em5.ControlNodes".ManualInput.sequence.status.seqActive;
   #statTonTimer[101].TON(IN := ("Unit1.Em5.ControlNodes".ManualInput.sequence.status.currentStep = #JOB_2_STEP_01) AND "Unit1.Em5.ControlNodes".ManualInput.sequence.status.seqActive AND "Unit1.Em5.ControlNodes".ManualInput."step".transition[201],
                          PT := #SeqNoDelayTime);
   IF #statTonTimer[101].Q THEN
       "Unit1.Em5.ControlNodes".ManualInput.sequence.status.nextStep := #JOB_2_STEP_11;
   END_IF;
END_REGION

REGION Network 16: Step[211] : Ng And Manual Input Cylinder WorkPos Command
   RUNG wire#powerrail
      { S7_Templates := "SrcType := DInt" } EQ_Contact(in1 := "Unit1.Em5.ControlNodes".ManualInput.sequence.status.currentStep, in2 := #JOB_2_STEP_11)
      Contact( "Unit1.Em5.ControlNodes".ManualInput.sequence.status.seqActive )
      wire#w1
      I_Contact( "Unit1.Em5.ControlNodes".cmNgAndManualInputCylinderUpDown.monitoring.inWorkPos )
      Coil( "Unit1.Em5.ControlNodes".ManualInput."step".action[211] )
   END_RUNG
   RUNG wire#w1
      Contact( "Unit1.Em5.ControlNodes".cmNgAndManualInputCylinderUpDown.monitoring.inWorkPos )
      Coil( "Unit1.Em5.ControlNodes".ManualInput."step".transition[211] )
   END_RUNG
   RUNG wire#w1
      Contact( "Unit1.Em5.ControlNodes".ManualInput."step".transition[211] )
      { S7_Templates := "time_type := Time" } #statTonTimer[211].TON(pt := #SeqDelayTime, et =>)
      Move(in := #JOB_2_STEP_21, out1 => "Unit1.Em5.ControlNodes".ManualInput.sequence.status.nextStep)
   END_RUNG
   // the same network as SCL:
   #_w1 := ("Unit1.Em5.ControlNodes".ManualInput.sequence.status.currentStep = #JOB_2_STEP_11) AND "Unit1.Em5.ControlNodes".ManualInput.sequence.status.seqActive;
   "Unit1.Em5.ControlNodes".ManualInput."step".action[211] := #_w1 AND NOT "Unit1.Em5.ControlNodes".cmNgAndManualInputCylinderUpDown.monitoring.inWorkPos;
   "Unit1.Em5.ControlNodes".ManualInput."step".transition[211] := #_w1 AND "Unit1.Em5.ControlNodes".cmNgAndManualInputCylinderUpDown.monitoring.inWorkPos;
   #statTonTimer[211].TON(IN := #_w1 AND "Unit1.Em5.ControlNodes".ManualInput."step".transition[211],
                          PT := #SeqDelayTime);
   IF #statTonTimer[211].Q THEN
       "Unit1.Em5.ControlNodes".ManualInput.sequence.status.nextStep := #JOB_2_STEP_21;
   END_IF;
END_REGION

REGION Network 17: Step[221] : Ng And Manual Input Vacuum WorkPos Command
   RUNG wire#powerrail
      { S7_Templates := "SrcType := DInt" } EQ_Contact(in1 := "Unit1.Em5.ControlNodes".ManualInput.sequence.status.currentStep, in2 := #JOB_2_STEP_21)
      Contact( "Unit1.Em5.ControlNodes".ManualInput.sequence.status.seqActive )
      wire#w1
      I_Contact( "Unit1.Em5.ControlNodes".cmNgAndManualInputVacuum1OnOff.monitoring.inWorkPos )
      Coil( "Unit1.Em5.ControlNodes".ManualInput."step".action[221] )
   END_RUNG
   RUNG wire#w1
      I_Contact( "Unit1.Em5.ControlNodes".cmNgAndManualInputVacuum2OnOff.monitoring.inWorkPos )
      Coil( "Unit1.Em5.ControlNodes".ManualInput."step".action[222] )
   END_RUNG
   RUNG wire#w1
      Contact( "Unit1.Em5.ControlNodes".cmNgAndManualInputVacuum1OnOff.monitoring.inWorkPos )
      Contact( "Unit1.Em5.ControlNodes".cmNgAndManualInputVacuum2OnOff.monitoring.inWorkPos )
      Coil( "Unit1.Em5.ControlNodes".ManualInput."step".transition[221] )
   END_RUNG
   RUNG wire#w1
      Contact( "Unit1.Em5.ControlNodes".ManualInput."step".transition[221] )
      { S7_Templates := "time_type := Time" } #statTonTimer[221].TON(pt := #SeqDelayTime, et =>)
      Move(in := #JOB_2_STEP_31, out1 => "Unit1.Em5.ControlNodes".ManualInput.sequence.status.nextStep)
   END_RUNG
   // the same network as SCL:
   #_w1 := ("Unit1.Em5.ControlNodes".ManualInput.sequence.status.currentStep = #JOB_2_STEP_21) AND "Unit1.Em5.ControlNodes".ManualInput.sequence.status.seqActive;
   "Unit1.Em5.ControlNodes".ManualInput."step".action[221] := #_w1 AND NOT "Unit1.Em5.ControlNodes".cmNgAndManualInputVacuum1OnOff.monitoring.inWorkPos;
   "Unit1.Em5.ControlNodes".ManualInput."step".action[222] := #_w1 AND NOT "Unit1.Em5.ControlNodes".cmNgAndManualInputVacuum2OnOff.monitoring.inWorkPos;
   "Unit1.Em5.ControlNodes".ManualInput."step".transition[221] := #_w1 AND "Unit1.Em5.ControlNodes".cmNgAndManualInputVacuum1OnOff.monitoring.inWorkPos AND "Unit1.Em5.ControlNodes".cmNgAndManualInputVacuum2OnOff.monitoring.inWorkPos;
   #statTonTimer[221].TON(IN := #_w1 AND "Unit1.Em5.ControlNodes".ManualInput."step".transition[221],
                          PT := #SeqDelayTime);
   IF #statTonTimer[221].Q THEN
       "Unit1.Em5.ControlNodes".ManualInput.sequence.status.nextStep := #JOB_2_STEP_31;
   END_IF;
END_REGION

REGION Network 18: Step[231] : Vibrator WorkPos Command
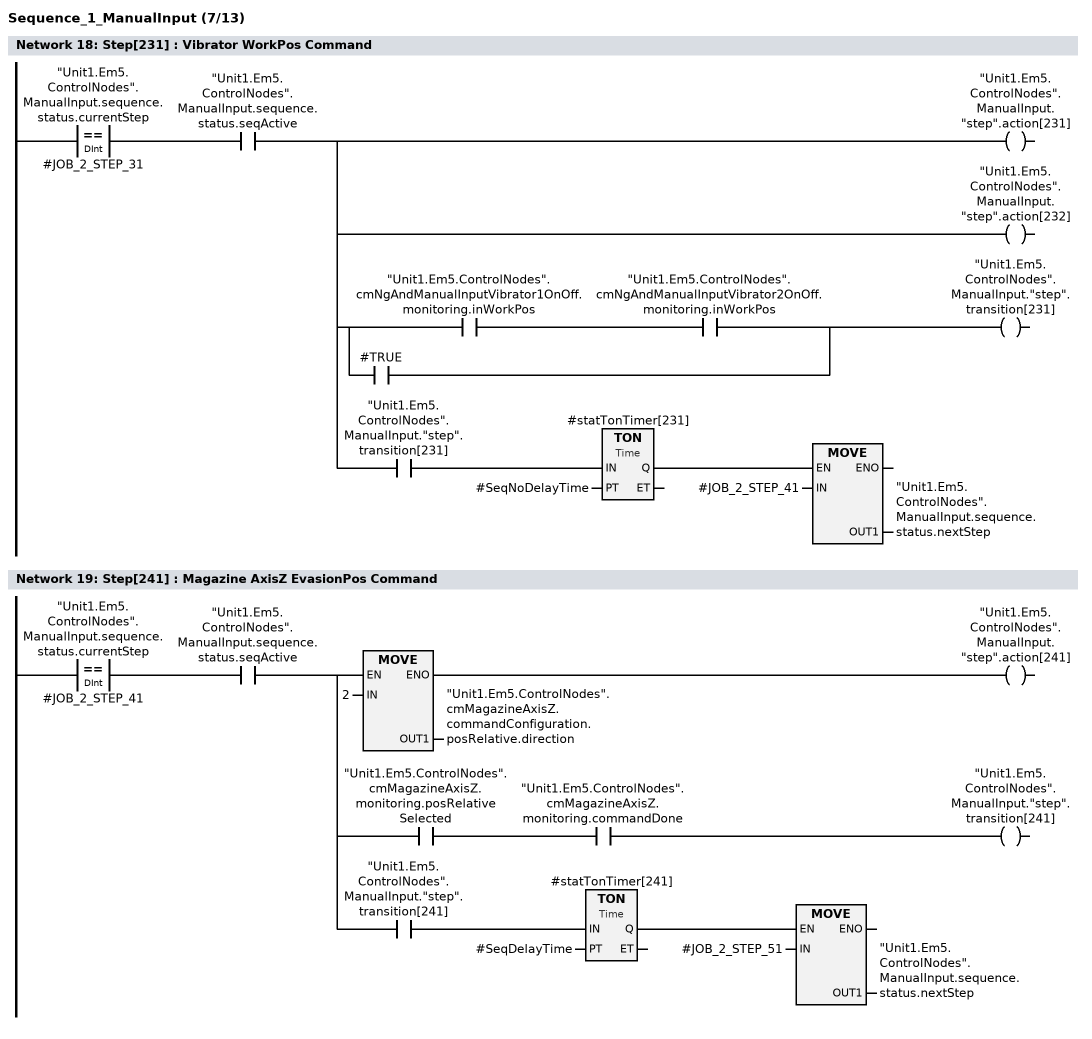
   RUNG wire#powerrail
      { S7_Templates := "SrcType := DInt" } EQ_Contact(in1 := "Unit1.Em5.ControlNodes".ManualInput.sequence.status.currentStep, in2 := #JOB_2_STEP_31)
      Contact( "Unit1.Em5.ControlNodes".ManualInput.sequence.status.seqActive )
      wire#w1
      Coil( "Unit1.Em5.ControlNodes".ManualInput."step".action[231] )
   END_RUNG
   RUNG wire#w1
      Coil( "Unit1.Em5.ControlNodes".ManualInput."step".action[232] )
   END_RUNG
   RUNG wire#w1
      Contact( "Unit1.Em5.ControlNodes".cmNgAndManualInputVibrator1OnOff.monitoring.inWorkPos )
      Contact( "Unit1.Em5.ControlNodes".cmNgAndManualInputVibrator2OnOff.monitoring.inWorkPos )
      wire#w2
      Coil( "Unit1.Em5.ControlNodes".ManualInput."step".transition[231] )
   END_RUNG
   RUNG wire#w1
      Contact( #TRUE )
   END_RUNG wire#w2
   RUNG wire#w1
      Contact( "Unit1.Em5.ControlNodes".ManualInput."step".transition[231] )
      { S7_Templates := "time_type := Time" } #statTonTimer[231].TON(pt := #SeqNoDelayTime, et =>)
      Move(in := #JOB_2_STEP_41, out1 => "Unit1.Em5.ControlNodes".ManualInput.sequence.status.nextStep)
   END_RUNG
   // the same network as SCL:
   "Unit1.Em5.ControlNodes".ManualInput."step".action[231] := ("Unit1.Em5.ControlNodes".ManualInput.sequence.status.currentStep = #JOB_2_STEP_31) AND "Unit1.Em5.ControlNodes".ManualInput.sequence.status.seqActive;
   "Unit1.Em5.ControlNodes".ManualInput."step".action[232] := ("Unit1.Em5.ControlNodes".ManualInput.sequence.status.currentStep = #JOB_2_STEP_31) AND "Unit1.Em5.ControlNodes".ManualInput.sequence.status.seqActive;
   "Unit1.Em5.ControlNodes".ManualInput."step".transition[231] := ("Unit1.Em5.ControlNodes".ManualInput.sequence.status.currentStep = #JOB_2_STEP_31) AND "Unit1.Em5.ControlNodes".ManualInput.sequence.status.seqActive AND (("Unit1.Em5.ControlNodes".cmNgAndManualInputVibrator1OnOff.monitoring.inWorkPos AND "Unit1.Em5.ControlNodes".cmNgAndManualInputVibrator2OnOff.monitoring.inWorkPos) OR #TRUE);
   #statTonTimer[231].TON(IN := ("Unit1.Em5.ControlNodes".ManualInput.sequence.status.currentStep = #JOB_2_STEP_31) AND "Unit1.Em5.ControlNodes".ManualInput.sequence.status.seqActive AND "Unit1.Em5.ControlNodes".ManualInput."step".transition[231],
                          PT := #SeqNoDelayTime);
   IF #statTonTimer[231].Q THEN
       "Unit1.Em5.ControlNodes".ManualInput.sequence.status.nextStep := #JOB_2_STEP_41;
   END_IF;
END_REGION

REGION Network 19: Step[241] : Magazine AxisZ EvasionPos Command
   RUNG wire#powerrail
      { S7_Templates := "SrcType := DInt" } EQ_Contact(in1 := "Unit1.Em5.ControlNodes".ManualInput.sequence.status.currentStep, in2 := #JOB_2_STEP_41)
      Contact( "Unit1.Em5.ControlNodes".ManualInput.sequence.status.seqActive )
      wire#w1
      Move(in := 2, out1 => "Unit1.Em5.ControlNodes".cmMagazineAxisZ.commandConfiguration.posRelative.direction)
      Coil( "Unit1.Em5.ControlNodes".ManualInput."step".action[241] )
   END_RUNG
   RUNG wire#w1
      Contact( "Unit1.Em5.ControlNodes".cmMagazineAxisZ.monitoring.posRelativeSelected )
      Contact( "Unit1.Em5.ControlNodes".cmMagazineAxisZ.monitoring.commandDone )
      Coil( "Unit1.Em5.ControlNodes".ManualInput."step".transition[241] )
   END_RUNG
   RUNG wire#w1
      Contact( "Unit1.Em5.ControlNodes".ManualInput."step".transition[241] )
      { S7_Templates := "time_type := Time" } #statTonTimer[241].TON(pt := #SeqDelayTime, et =>)
      Move(in := #JOB_2_STEP_51, out1 => "Unit1.Em5.ControlNodes".ManualInput.sequence.status.nextStep)
   END_RUNG
   // the same network as SCL:
   #_w1 := ("Unit1.Em5.ControlNodes".ManualInput.sequence.status.currentStep = #JOB_2_STEP_41) AND "Unit1.Em5.ControlNodes".ManualInput.sequence.status.seqActive;
   IF #_w1 THEN
       "Unit1.Em5.ControlNodes".cmMagazineAxisZ.commandConfiguration.posRelative.direction := 2;
   END_IF;
   "Unit1.Em5.ControlNodes".ManualInput."step".action[241] := #_w1;
   "Unit1.Em5.ControlNodes".ManualInput."step".transition[241] := #_w1 AND "Unit1.Em5.ControlNodes".cmMagazineAxisZ.monitoring.posRelativeSelected AND "Unit1.Em5.ControlNodes".cmMagazineAxisZ.monitoring.commandDone;
   #statTonTimer[241].TON(IN := #_w1 AND "Unit1.Em5.ControlNodes".ManualInput."step".transition[241],
                          PT := #SeqDelayTime);
   IF #statTonTimer[241].Q THEN
       "Unit1.Em5.ControlNodes".ManualInput.sequence.status.nextStep := #JOB_2_STEP_51;
   END_IF;
END_REGION

REGION Network 20: Step[251] : Vibrator HomePos Command
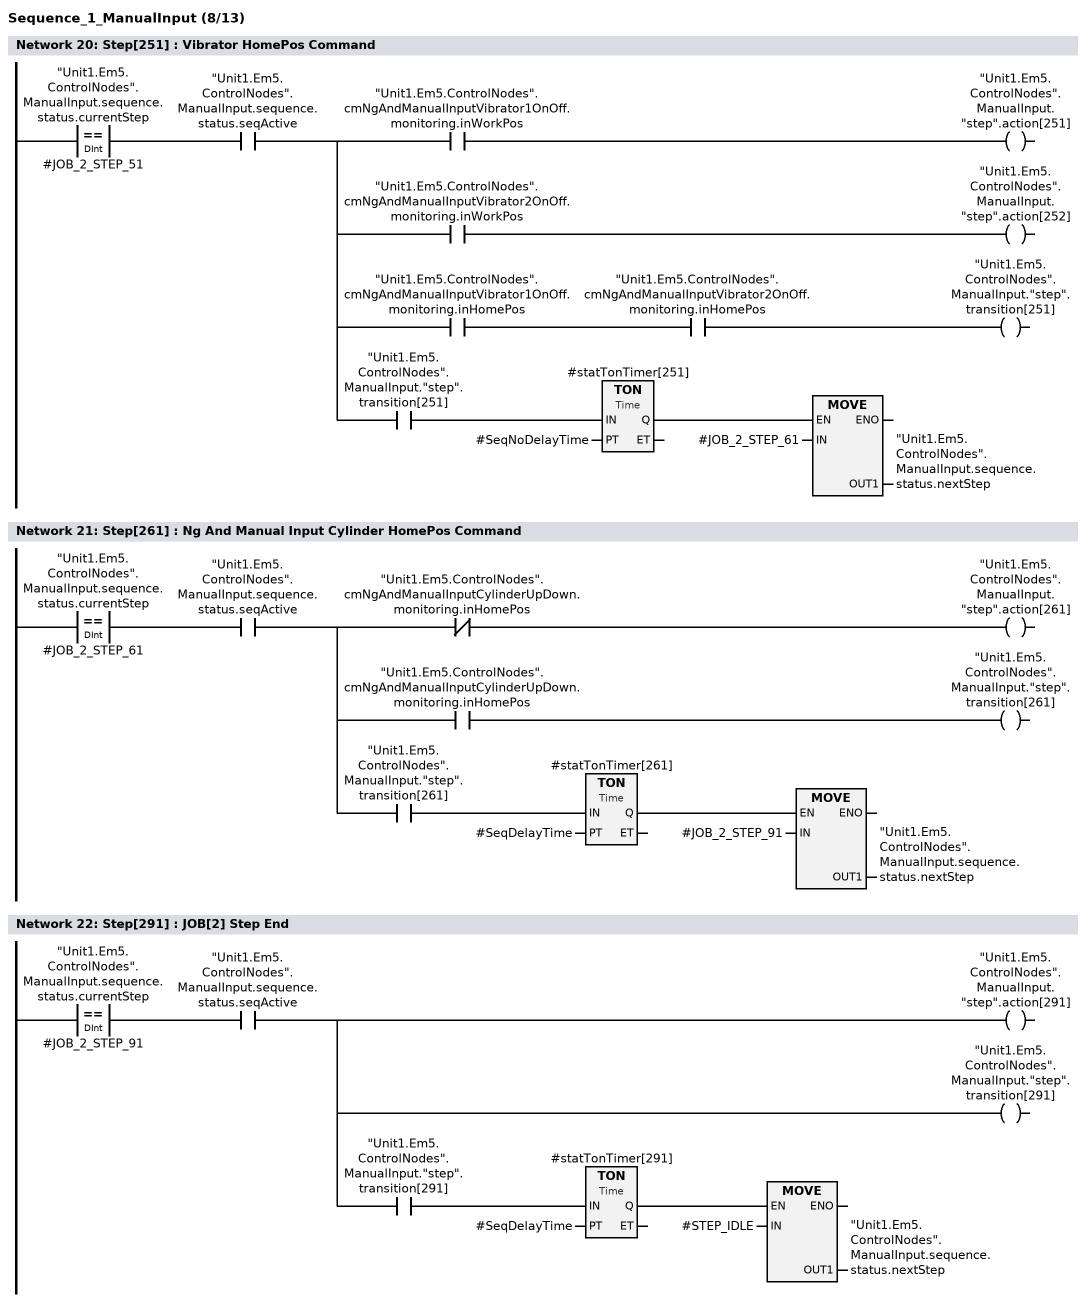
   RUNG wire#powerrail
      { S7_Templates := "SrcType := DInt" } EQ_Contact(in1 := "Unit1.Em5.ControlNodes".ManualInput.sequence.status.currentStep, in2 := #JOB_2_STEP_51)
      Contact( "Unit1.Em5.ControlNodes".ManualInput.sequence.status.seqActive )
      wire#w1
      Contact( "Unit1.Em5.ControlNodes".cmNgAndManualInputVibrator1OnOff.monitoring.inWorkPos )
      Coil( "Unit1.Em5.ControlNodes".ManualInput."step".action[251] )
   END_RUNG
   RUNG wire#w1
      Contact( "Unit1.Em5.ControlNodes".cmNgAndManualInputVibrator2OnOff.monitoring.inWorkPos )
      Coil( "Unit1.Em5.ControlNodes".ManualInput."step".action[252] )
   END_RUNG
   RUNG wire#w1
      Contact( "Unit1.Em5.ControlNodes".cmNgAndManualInputVibrator1OnOff.monitoring.inHomePos )
      Contact( "Unit1.Em5.ControlNodes".cmNgAndManualInputVibrator2OnOff.monitoring.inHomePos )
      Coil( "Unit1.Em5.ControlNodes".ManualInput."step".transition[251] )
   END_RUNG
   RUNG wire#w1
      Contact( "Unit1.Em5.ControlNodes".ManualInput."step".transition[251] )
      { S7_Templates := "time_type := Time" } #statTonTimer[251].TON(pt := #SeqNoDelayTime, et =>)
      Move(in := #JOB_2_STEP_61, out1 => "Unit1.Em5.ControlNodes".ManualInput.sequence.status.nextStep)
   END_RUNG
   // the same network as SCL:
   #_w1 := ("Unit1.Em5.ControlNodes".ManualInput.sequence.status.currentStep = #JOB_2_STEP_51) AND "Unit1.Em5.ControlNodes".ManualInput.sequence.status.seqActive;
   "Unit1.Em5.ControlNodes".ManualInput."step".action[251] := #_w1 AND "Unit1.Em5.ControlNodes".cmNgAndManualInputVibrator1OnOff.monitoring.inWorkPos;
   "Unit1.Em5.ControlNodes".ManualInput."step".action[252] := #_w1 AND "Unit1.Em5.ControlNodes".cmNgAndManualInputVibrator2OnOff.monitoring.inWorkPos;
   "Unit1.Em5.ControlNodes".ManualInput."step".transition[251] := #_w1 AND "Unit1.Em5.ControlNodes".cmNgAndManualInputVibrator1OnOff.monitoring.inHomePos AND "Unit1.Em5.ControlNodes".cmNgAndManualInputVibrator2OnOff.monitoring.inHomePos;
   #statTonTimer[251].TON(IN := #_w1 AND "Unit1.Em5.ControlNodes".ManualInput."step".transition[251],
                          PT := #SeqNoDelayTime);
   IF #statTonTimer[251].Q THEN
       "Unit1.Em5.ControlNodes".ManualInput.sequence.status.nextStep := #JOB_2_STEP_61;
   END_IF;
END_REGION

REGION Network 21: Step[261] : Ng And Manual Input Cylinder HomePos Command
   RUNG wire#powerrail
      { S7_Templates := "SrcType := DInt" } EQ_Contact(in1 := "Unit1.Em5.ControlNodes".ManualInput.sequence.status.currentStep, in2 := #JOB_2_STEP_61)
      Contact( "Unit1.Em5.ControlNodes".ManualInput.sequence.status.seqActive )
      wire#w1
      I_Contact( "Unit1.Em5.ControlNodes".cmNgAndManualInputCylinderUpDown.monitoring.inHomePos )
      Coil( "Unit1.Em5.ControlNodes".ManualInput."step".action[261] )
   END_RUNG
   RUNG wire#w1
      Contact( "Unit1.Em5.ControlNodes".cmNgAndManualInputCylinderUpDown.monitoring.inHomePos )
      Coil( "Unit1.Em5.ControlNodes".ManualInput."step".transition[261] )
   END_RUNG
   RUNG wire#w1
      Contact( "Unit1.Em5.ControlNodes".ManualInput."step".transition[261] )
      { S7_Templates := "time_type := Time" } #statTonTimer[261].TON(pt := #SeqDelayTime, et =>)
      Move(in := #JOB_2_STEP_91, out1 => "Unit1.Em5.ControlNodes".ManualInput.sequence.status.nextStep)
   END_RUNG
   // the same network as SCL:
   #_w1 := ("Unit1.Em5.ControlNodes".ManualInput.sequence.status.currentStep = #JOB_2_STEP_61) AND "Unit1.Em5.ControlNodes".ManualInput.sequence.status.seqActive;
   "Unit1.Em5.ControlNodes".ManualInput."step".action[261] := #_w1 AND NOT "Unit1.Em5.ControlNodes".cmNgAndManualInputCylinderUpDown.monitoring.inHomePos;
   "Unit1.Em5.ControlNodes".ManualInput."step".transition[261] := #_w1 AND "Unit1.Em5.ControlNodes".cmNgAndManualInputCylinderUpDown.monitoring.inHomePos;
   #statTonTimer[261].TON(IN := #_w1 AND "Unit1.Em5.ControlNodes".ManualInput."step".transition[261],
                          PT := #SeqDelayTime);
   IF #statTonTimer[261].Q THEN
       "Unit1.Em5.ControlNodes".ManualInput.sequence.status.nextStep := #JOB_2_STEP_91;
   END_IF;
END_REGION

REGION Network 22: Step[291] : JOB[2] Step End
   RUNG wire#powerrail
      { S7_Templates := "SrcType := DInt" } EQ_Contact(in1 := "Unit1.Em5.ControlNodes".ManualInput.sequence.status.currentStep, in2 := #JOB_2_STEP_91)
      Contact( "Unit1.Em5.ControlNodes".ManualInput.sequence.status.seqActive )
      wire#w1
      Coil( "Unit1.Em5.ControlNodes".ManualInput."step".action[291] )
   END_RUNG
   RUNG wire#w1
      Coil( "Unit1.Em5.ControlNodes".ManualInput."step".transition[291] )
   END_RUNG
   RUNG wire#w1
      Contact( "Unit1.Em5.ControlNodes".ManualInput."step".transition[291] )
      { S7_Templates := "time_type := Time" } #statTonTimer[291].TON(pt := #SeqDelayTime, et =>)
      Move(in := #STEP_IDLE, out1 => "Unit1.Em5.ControlNodes".ManualInput.sequence.status.nextStep)
   END_RUNG
   // the same network as SCL:
   "Unit1.Em5.ControlNodes".ManualInput."step".action[291] := ("Unit1.Em5.ControlNodes".ManualInput.sequence.status.currentStep = #JOB_2_STEP_91) AND "Unit1.Em5.ControlNodes".ManualInput.sequence.status.seqActive;
   "Unit1.Em5.ControlNodes".ManualInput."step".transition[291] := ("Unit1.Em5.ControlNodes".ManualInput.sequence.status.currentStep = #JOB_2_STEP_91) AND "Unit1.Em5.ControlNodes".ManualInput.sequence.status.seqActive;
   #statTonTimer[291].TON(IN := ("Unit1.Em5.ControlNodes".ManualInput.sequence.status.currentStep = #JOB_2_STEP_91) AND "Unit1.Em5.ControlNodes".ManualInput.sequence.status.seqActive AND "Unit1.Em5.ControlNodes".ManualInput."step".transition[291],
                          PT := #SeqDelayTime);
   IF #statTonTimer[291].Q THEN
       "Unit1.Em5.ControlNodes".ManualInput.sequence.status.nextStep := #STEP_IDLE;
   END_IF;
END_REGION

REGION Network 23: ******************** JOB[3] UNLOADING AUTO ********************
END_REGION

REGION Network 24: Step[301] : JOB[3] Condition
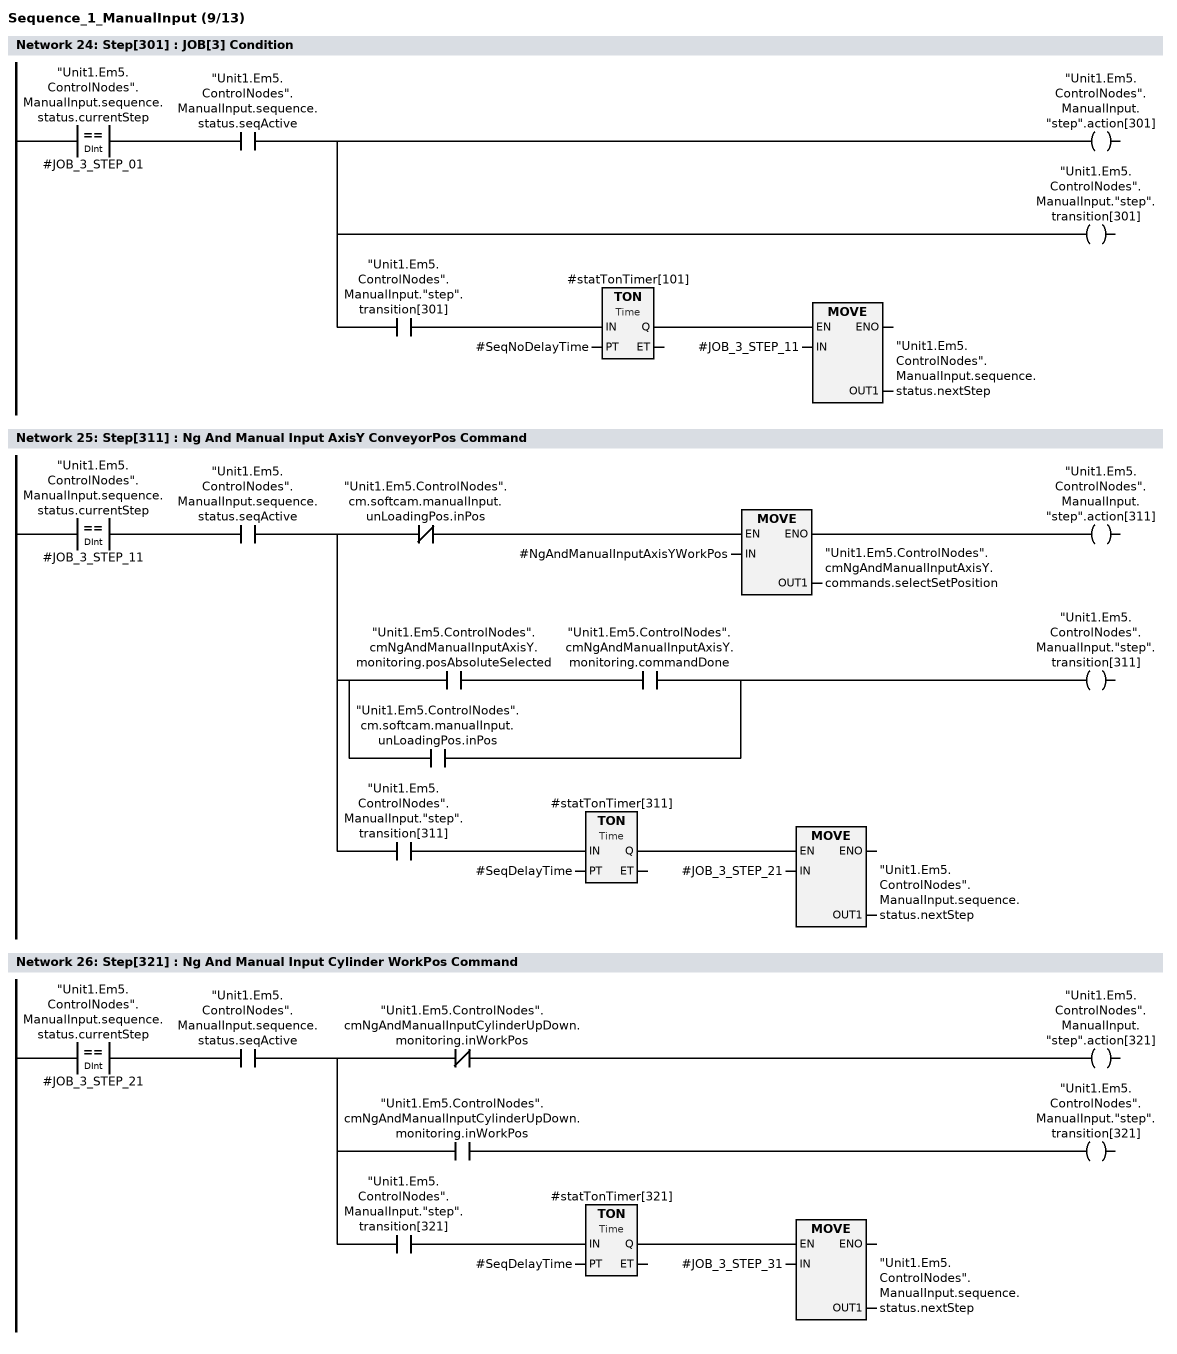
   RUNG wire#powerrail
      { S7_Templates := "SrcType := DInt" } EQ_Contact(in1 := "Unit1.Em5.ControlNodes".ManualInput.sequence.status.currentStep, in2 := #JOB_3_STEP_01)
      Contact( "Unit1.Em5.ControlNodes".ManualInput.sequence.status.seqActive )
      wire#w1
      Coil( "Unit1.Em5.ControlNodes".ManualInput."step".action[301] )
   END_RUNG
   RUNG wire#w1
      Coil( "Unit1.Em5.ControlNodes".ManualInput."step".transition[301] )
   END_RUNG
   RUNG wire#w1
      Contact( "Unit1.Em5.ControlNodes".ManualInput."step".transition[301] )
      { S7_Templates := "time_type := Time" } #statTonTimer[101].TON(pt := #SeqNoDelayTime, et =>)
      Move(in := #JOB_3_STEP_11, out1 => "Unit1.Em5.ControlNodes".ManualInput.sequence.status.nextStep)
   END_RUNG
   // the same network as SCL:
   "Unit1.Em5.ControlNodes".ManualInput."step".action[301] := ("Unit1.Em5.ControlNodes".ManualInput.sequence.status.currentStep = #JOB_3_STEP_01) AND "Unit1.Em5.ControlNodes".ManualInput.sequence.status.seqActive;
   "Unit1.Em5.ControlNodes".ManualInput."step".transition[301] := ("Unit1.Em5.ControlNodes".ManualInput.sequence.status.currentStep = #JOB_3_STEP_01) AND "Unit1.Em5.ControlNodes".ManualInput.sequence.status.seqActive;
   #statTonTimer[101].TON(IN := ("Unit1.Em5.ControlNodes".ManualInput.sequence.status.currentStep = #JOB_3_STEP_01) AND "Unit1.Em5.ControlNodes".ManualInput.sequence.status.seqActive AND "Unit1.Em5.ControlNodes".ManualInput."step".transition[301],
                          PT := #SeqNoDelayTime);
   IF #statTonTimer[101].Q THEN
       "Unit1.Em5.ControlNodes".ManualInput.sequence.status.nextStep := #JOB_3_STEP_11;
   END_IF;
END_REGION

REGION Network 25: Step[311] : Ng And Manual Input AxisY ConveyorPos Command
   RUNG wire#powerrail
      { S7_Templates := "SrcType := DInt" } EQ_Contact(in1 := "Unit1.Em5.ControlNodes".ManualInput.sequence.status.currentStep, in2 := #JOB_3_STEP_11)
      Contact( "Unit1.Em5.ControlNodes".ManualInput.sequence.status.seqActive )
      wire#w1
      I_Contact( "Unit1.Em5.ControlNodes".cm.softcam.manualInput.unLoadingPos.inPos )
      Move(in := #NgAndManualInputAxisYWorkPos, out1 => "Unit1.Em5.ControlNodes".cmNgAndManualInputAxisY.commands.selectSetPosition)
      Coil( "Unit1.Em5.ControlNodes".ManualInput."step".action[311] )
   END_RUNG
   RUNG wire#w1
      Contact( "Unit1.Em5.ControlNodes".cmNgAndManualInputAxisY.monitoring.posAbsoluteSelected )
      Contact( "Unit1.Em5.ControlNodes".cmNgAndManualInputAxisY.monitoring.commandDone )
      wire#w2
      Coil( "Unit1.Em5.ControlNodes".ManualInput."step".transition[311] )
   END_RUNG
   RUNG wire#w1
      Contact( "Unit1.Em5.ControlNodes".cm.softcam.manualInput.unLoadingPos.inPos )
   END_RUNG wire#w2
   RUNG wire#w1
      Contact( "Unit1.Em5.ControlNodes".ManualInput."step".transition[311] )
      { S7_Templates := "time_type := Time" } #statTonTimer[311].TON(pt := #SeqDelayTime, et =>)
      Move(in := #JOB_3_STEP_21, out1 => "Unit1.Em5.ControlNodes".ManualInput.sequence.status.nextStep)
   END_RUNG
   // the same network as SCL:
   #_w1 := ("Unit1.Em5.ControlNodes".ManualInput.sequence.status.currentStep = #JOB_3_STEP_11) AND "Unit1.Em5.ControlNodes".ManualInput.sequence.status.seqActive;
   #_w2 := #_w1 AND NOT "Unit1.Em5.ControlNodes".cm.softcam.manualInput.unLoadingPos.inPos;
   IF #_w2 THEN
       "Unit1.Em5.ControlNodes".cmNgAndManualInputAxisY.commands.selectSetPosition := #NgAndManualInputAxisYWorkPos;
   END_IF;
   "Unit1.Em5.ControlNodes".ManualInput."step".action[311] := #_w2;
   "Unit1.Em5.ControlNodes".ManualInput."step".transition[311] := #_w1 AND (("Unit1.Em5.ControlNodes".cmNgAndManualInputAxisY.monitoring.posAbsoluteSelected AND "Unit1.Em5.ControlNodes".cmNgAndManualInputAxisY.monitoring.commandDone) OR "Unit1.Em5.ControlNodes".cm.softcam.manualInput.unLoadingPos.inPos);
   #statTonTimer[311].TON(IN := #_w1 AND "Unit1.Em5.ControlNodes".ManualInput."step".transition[311],
                          PT := #SeqDelayTime);
   IF #statTonTimer[311].Q THEN
       "Unit1.Em5.ControlNodes".ManualInput.sequence.status.nextStep := #JOB_3_STEP_21;
   END_IF;
END_REGION

REGION Network 26: Step[321] : Ng And Manual Input Cylinder WorkPos Command
   RUNG wire#powerrail
      { S7_Templates := "SrcType := DInt" } EQ_Contact(in1 := "Unit1.Em5.ControlNodes".ManualInput.sequence.status.currentStep, in2 := #JOB_3_STEP_21)
      Contact( "Unit1.Em5.ControlNodes".ManualInput.sequence.status.seqActive )
      wire#w1
      I_Contact( "Unit1.Em5.ControlNodes".cmNgAndManualInputCylinderUpDown.monitoring.inWorkPos )
      Coil( "Unit1.Em5.ControlNodes".ManualInput."step".action[321] )
   END_RUNG
   RUNG wire#w1
      Contact( "Unit1.Em5.ControlNodes".cmNgAndManualInputCylinderUpDown.monitoring.inWorkPos )
      Coil( "Unit1.Em5.ControlNodes".ManualInput."step".transition[321] )
   END_RUNG
   RUNG wire#w1
      Contact( "Unit1.Em5.ControlNodes".ManualInput."step".transition[321] )
      { S7_Templates := "time_type := Time" } #statTonTimer[321].TON(pt := #SeqDelayTime, et =>)
      Move(in := #JOB_3_STEP_31, out1 => "Unit1.Em5.ControlNodes".ManualInput.sequence.status.nextStep)
   END_RUNG
   // the same network as SCL:
   #_w1 := ("Unit1.Em5.ControlNodes".ManualInput.sequence.status.currentStep = #JOB_3_STEP_21) AND "Unit1.Em5.ControlNodes".ManualInput.sequence.status.seqActive;
   "Unit1.Em5.ControlNodes".ManualInput."step".action[321] := #_w1 AND NOT "Unit1.Em5.ControlNodes".cmNgAndManualInputCylinderUpDown.monitoring.inWorkPos;
   "Unit1.Em5.ControlNodes".ManualInput."step".transition[321] := #_w1 AND "Unit1.Em5.ControlNodes".cmNgAndManualInputCylinderUpDown.monitoring.inWorkPos;
   #statTonTimer[321].TON(IN := #_w1 AND "Unit1.Em5.ControlNodes".ManualInput."step".transition[321],
                          PT := #SeqDelayTime);
   IF #statTonTimer[321].Q THEN
       "Unit1.Em5.ControlNodes".ManualInput.sequence.status.nextStep := #JOB_3_STEP_31;
   END_IF;
END_REGION

REGION Network 27: Step[331] : Ng And Manual Input Vacuum HomePos Command
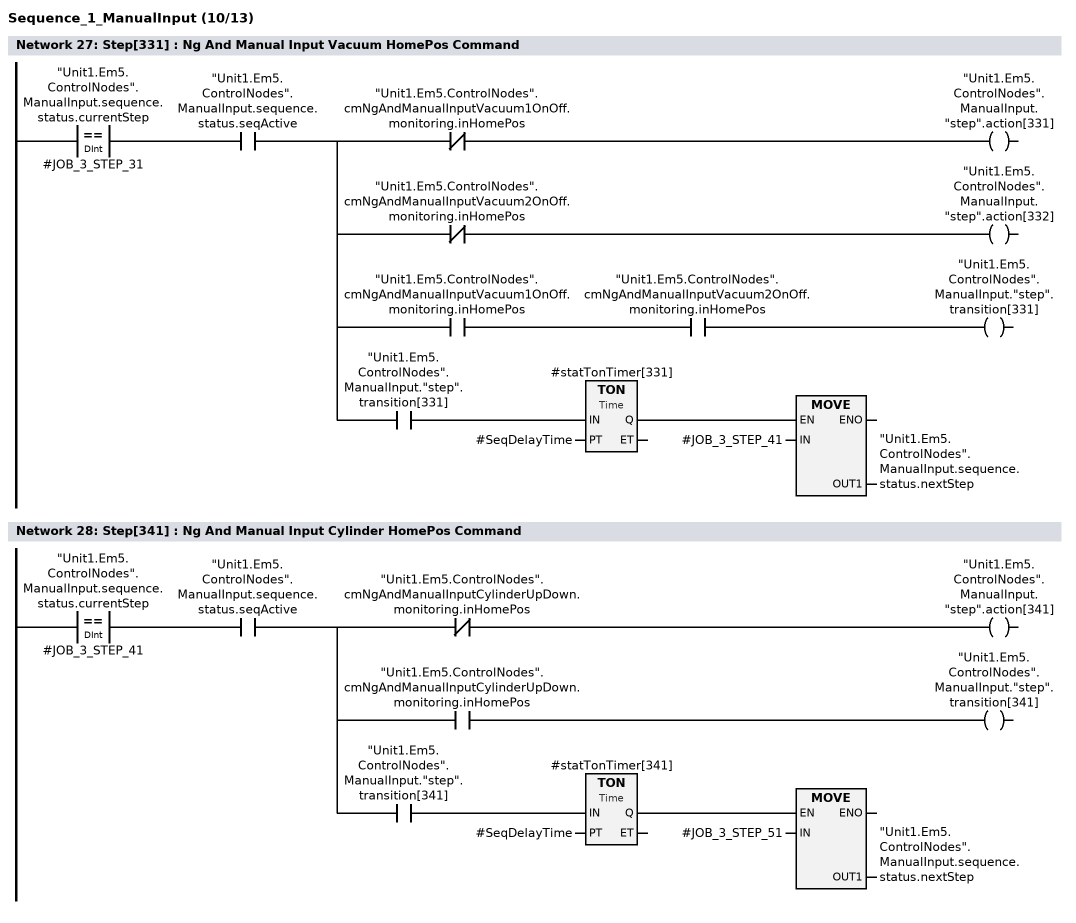
   RUNG wire#powerrail
      { S7_Templates := "SrcType := DInt" } EQ_Contact(in1 := "Unit1.Em5.ControlNodes".ManualInput.sequence.status.currentStep, in2 := #JOB_3_STEP_31)
      Contact( "Unit1.Em5.ControlNodes".ManualInput.sequence.status.seqActive )
      wire#w1
      I_Contact( "Unit1.Em5.ControlNodes".cmNgAndManualInputVacuum1OnOff.monitoring.inHomePos )
      Coil( "Unit1.Em5.ControlNodes".ManualInput."step".action[331] )
   END_RUNG
   RUNG wire#w1
      I_Contact( "Unit1.Em5.ControlNodes".cmNgAndManualInputVacuum2OnOff.monitoring.inHomePos )
      Coil( "Unit1.Em5.ControlNodes".ManualInput."step".action[332] )
   END_RUNG
   RUNG wire#w1
      Contact( "Unit1.Em5.ControlNodes".cmNgAndManualInputVacuum1OnOff.monitoring.inHomePos )
      Contact( "Unit1.Em5.ControlNodes".cmNgAndManualInputVacuum2OnOff.monitoring.inHomePos )
      Coil( "Unit1.Em5.ControlNodes".ManualInput."step".transition[331] )
   END_RUNG
   RUNG wire#w1
      Contact( "Unit1.Em5.ControlNodes".ManualInput."step".transition[331] )
      { S7_Templates := "time_type := Time" } #statTonTimer[331].TON(pt := #SeqDelayTime, et =>)
      Move(in := #JOB_3_STEP_41, out1 => "Unit1.Em5.ControlNodes".ManualInput.sequence.status.nextStep)
   END_RUNG
   // the same network as SCL:
   #_w1 := ("Unit1.Em5.ControlNodes".ManualInput.sequence.status.currentStep = #JOB_3_STEP_31) AND "Unit1.Em5.ControlNodes".ManualInput.sequence.status.seqActive;
   "Unit1.Em5.ControlNodes".ManualInput."step".action[331] := #_w1 AND NOT "Unit1.Em5.ControlNodes".cmNgAndManualInputVacuum1OnOff.monitoring.inHomePos;
   "Unit1.Em5.ControlNodes".ManualInput."step".action[332] := #_w1 AND NOT "Unit1.Em5.ControlNodes".cmNgAndManualInputVacuum2OnOff.monitoring.inHomePos;
   "Unit1.Em5.ControlNodes".ManualInput."step".transition[331] := #_w1 AND "Unit1.Em5.ControlNodes".cmNgAndManualInputVacuum1OnOff.monitoring.inHomePos AND "Unit1.Em5.ControlNodes".cmNgAndManualInputVacuum2OnOff.monitoring.inHomePos;
   #statTonTimer[331].TON(IN := #_w1 AND "Unit1.Em5.ControlNodes".ManualInput."step".transition[331],
                          PT := #SeqDelayTime);
   IF #statTonTimer[331].Q THEN
       "Unit1.Em5.ControlNodes".ManualInput.sequence.status.nextStep := #JOB_3_STEP_41;
   END_IF;
END_REGION

REGION Network 28: Step[341] : Ng And Manual Input Cylinder HomePos Command
   RUNG wire#powerrail
      { S7_Templates := "SrcType := DInt" } EQ_Contact(in1 := "Unit1.Em5.ControlNodes".ManualInput.sequence.status.currentStep, in2 := #JOB_3_STEP_41)
      Contact( "Unit1.Em5.ControlNodes".ManualInput.sequence.status.seqActive )
      wire#w1
      I_Contact( "Unit1.Em5.ControlNodes".cmNgAndManualInputCylinderUpDown.monitoring.inHomePos )
      Coil( "Unit1.Em5.ControlNodes".ManualInput."step".action[341] )
   END_RUNG
   RUNG wire#w1
      Contact( "Unit1.Em5.ControlNodes".cmNgAndManualInputCylinderUpDown.monitoring.inHomePos )
      Coil( "Unit1.Em5.ControlNodes".ManualInput."step".transition[341] )
   END_RUNG
   RUNG wire#w1
      Contact( "Unit1.Em5.ControlNodes".ManualInput."step".transition[341] )
      { S7_Templates := "time_type := Time" } #statTonTimer[341].TON(pt := #SeqDelayTime, et =>)
      Move(in := #JOB_3_STEP_51, out1 => "Unit1.Em5.ControlNodes".ManualInput.sequence.status.nextStep)
   END_RUNG
   // the same network as SCL:
   #_w1 := ("Unit1.Em5.ControlNodes".ManualInput.sequence.status.currentStep = #JOB_3_STEP_41) AND "Unit1.Em5.ControlNodes".ManualInput.sequence.status.seqActive;
   "Unit1.Em5.ControlNodes".ManualInput."step".action[341] := #_w1 AND NOT "Unit1.Em5.ControlNodes".cmNgAndManualInputCylinderUpDown.monitoring.inHomePos;
   "Unit1.Em5.ControlNodes".ManualInput."step".transition[341] := #_w1 AND "Unit1.Em5.ControlNodes".cmNgAndManualInputCylinderUpDown.monitoring.inHomePos;
   #statTonTimer[341].TON(IN := #_w1 AND "Unit1.Em5.ControlNodes".ManualInput."step".transition[341],
                          PT := #SeqDelayTime);
   IF #statTonTimer[341].Q THEN
       "Unit1.Em5.ControlNodes".ManualInput.sequence.status.nextStep := #JOB_3_STEP_51;
   END_IF;
END_REGION

REGION Network 29: Step[351] : Ng And Manual Input AxisY HomePos Command
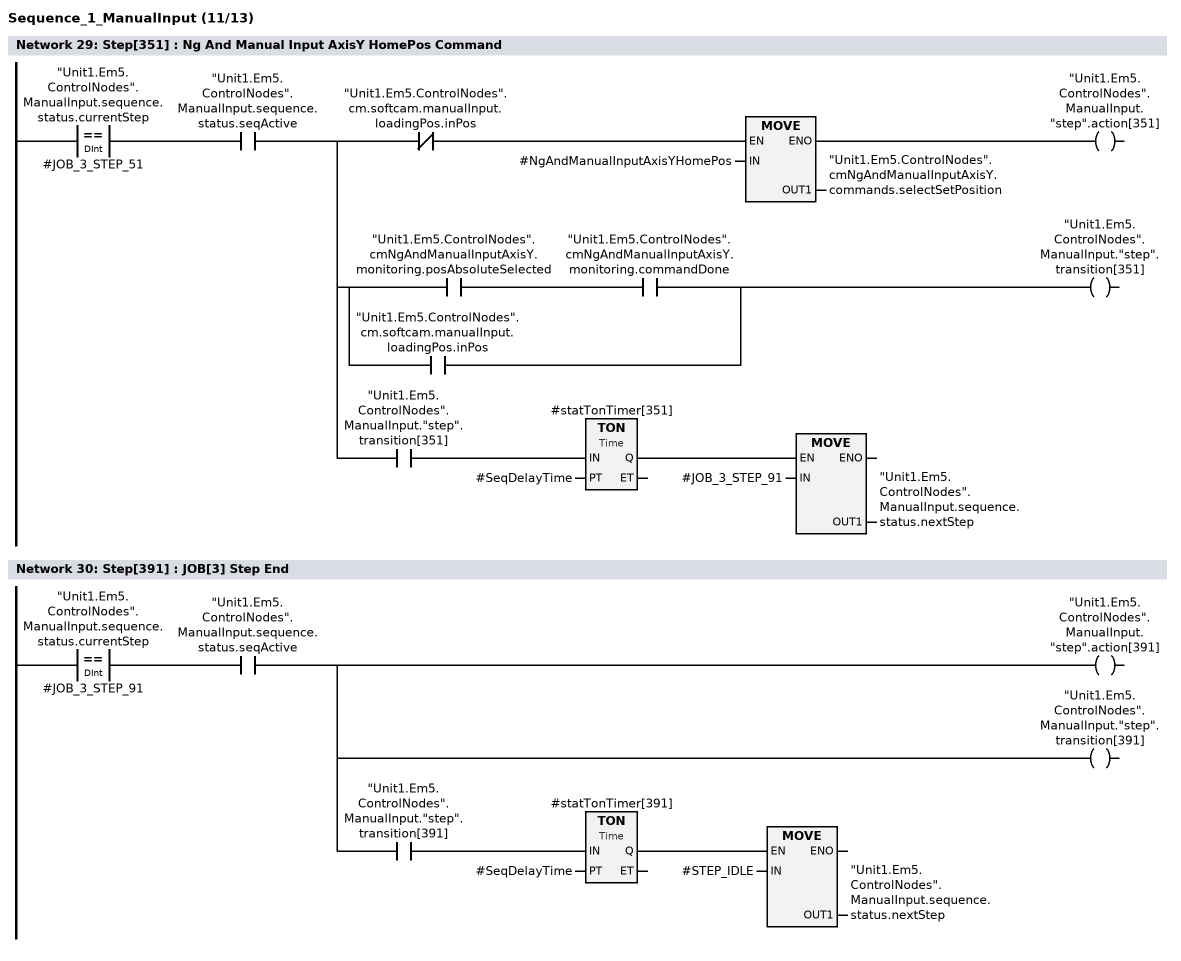
   RUNG wire#powerrail
      { S7_Templates := "SrcType := DInt" } EQ_Contact(in1 := "Unit1.Em5.ControlNodes".ManualInput.sequence.status.currentStep, in2 := #JOB_3_STEP_51)
      Contact( "Unit1.Em5.ControlNodes".ManualInput.sequence.status.seqActive )
      wire#w1
      I_Contact( "Unit1.Em5.ControlNodes".cm.softcam.manualInput.loadingPos.inPos )
      Move(in := #NgAndManualInputAxisYHomePos, out1 => "Unit1.Em5.ControlNodes".cmNgAndManualInputAxisY.commands.selectSetPosition)
      Coil( "Unit1.Em5.ControlNodes".ManualInput."step".action[351] )
   END_RUNG
   RUNG wire#w1
      Contact( "Unit1.Em5.ControlNodes".cmNgAndManualInputAxisY.monitoring.posAbsoluteSelected )
      Contact( "Unit1.Em5.ControlNodes".cmNgAndManualInputAxisY.monitoring.commandDone )
      wire#w2
      Coil( "Unit1.Em5.ControlNodes".ManualInput."step".transition[351] )
   END_RUNG
   RUNG wire#w1
      Contact( "Unit1.Em5.ControlNodes".cm.softcam.manualInput.loadingPos.inPos )
   END_RUNG wire#w2
   RUNG wire#w1
      Contact( "Unit1.Em5.ControlNodes".ManualInput."step".transition[351] )
      { S7_Templates := "time_type := Time" } #statTonTimer[351].TON(pt := #SeqDelayTime, et =>)
      Move(in := #JOB_3_STEP_91, out1 => "Unit1.Em5.ControlNodes".ManualInput.sequence.status.nextStep)
   END_RUNG
   // the same network as SCL:
   #_w1 := ("Unit1.Em5.ControlNodes".ManualInput.sequence.status.currentStep = #JOB_3_STEP_51) AND "Unit1.Em5.ControlNodes".ManualInput.sequence.status.seqActive;
   #_w2 := #_w1 AND NOT "Unit1.Em5.ControlNodes".cm.softcam.manualInput.loadingPos.inPos;
   IF #_w2 THEN
       "Unit1.Em5.ControlNodes".cmNgAndManualInputAxisY.commands.selectSetPosition := #NgAndManualInputAxisYHomePos;
   END_IF;
   "Unit1.Em5.ControlNodes".ManualInput."step".action[351] := #_w2;
   "Unit1.Em5.ControlNodes".ManualInput."step".transition[351] := #_w1 AND (("Unit1.Em5.ControlNodes".cmNgAndManualInputAxisY.monitoring.posAbsoluteSelected AND "Unit1.Em5.ControlNodes".cmNgAndManualInputAxisY.monitoring.commandDone) OR "Unit1.Em5.ControlNodes".cm.softcam.manualInput.loadingPos.inPos);
   #statTonTimer[351].TON(IN := #_w1 AND "Unit1.Em5.ControlNodes".ManualInput."step".transition[351],
                          PT := #SeqDelayTime);
   IF #statTonTimer[351].Q THEN
       "Unit1.Em5.ControlNodes".ManualInput.sequence.status.nextStep := #JOB_3_STEP_91;
   END_IF;
END_REGION

REGION Network 30: Step[391] : JOB[3] Step End
   RUNG wire#powerrail
      { S7_Templates := "SrcType := DInt" } EQ_Contact(in1 := "Unit1.Em5.ControlNodes".ManualInput.sequence.status.currentStep, in2 := #JOB_3_STEP_91)
      Contact( "Unit1.Em5.ControlNodes".ManualInput.sequence.status.seqActive )
      wire#w1
      Coil( "Unit1.Em5.ControlNodes".ManualInput."step".action[391] )
   END_RUNG
   RUNG wire#w1
      Coil( "Unit1.Em5.ControlNodes".ManualInput."step".transition[391] )
   END_RUNG
   RUNG wire#w1
      Contact( "Unit1.Em5.ControlNodes".ManualInput."step".transition[391] )
      { S7_Templates := "time_type := Time" } #statTonTimer[391].TON(pt := #SeqDelayTime, et =>)
      Move(in := #STEP_IDLE, out1 => "Unit1.Em5.ControlNodes".ManualInput.sequence.status.nextStep)
   END_RUNG
   // the same network as SCL:
   "Unit1.Em5.ControlNodes".ManualInput."step".action[391] := ("Unit1.Em5.ControlNodes".ManualInput.sequence.status.currentStep = #JOB_3_STEP_91) AND "Unit1.Em5.ControlNodes".ManualInput.sequence.status.seqActive;
   "Unit1.Em5.ControlNodes".ManualInput."step".transition[391] := ("Unit1.Em5.ControlNodes".ManualInput.sequence.status.currentStep = #JOB_3_STEP_91) AND "Unit1.Em5.ControlNodes".ManualInput.sequence.status.seqActive;
   #statTonTimer[391].TON(IN := ("Unit1.Em5.ControlNodes".ManualInput.sequence.status.currentStep = #JOB_3_STEP_91) AND "Unit1.Em5.ControlNodes".ManualInput.sequence.status.seqActive AND "Unit1.Em5.ControlNodes".ManualInput."step".transition[391],
                          PT := #SeqDelayTime);
   IF #statTonTimer[391].Q THEN
       "Unit1.Em5.ControlNodes".ManualInput.sequence.status.nextStep := #STEP_IDLE;
   END_IF;
END_REGION

REGION Network 31: *************** IMMEDIATE STOP ****************
END_REGION

REGION Network 32: Immediate Stop
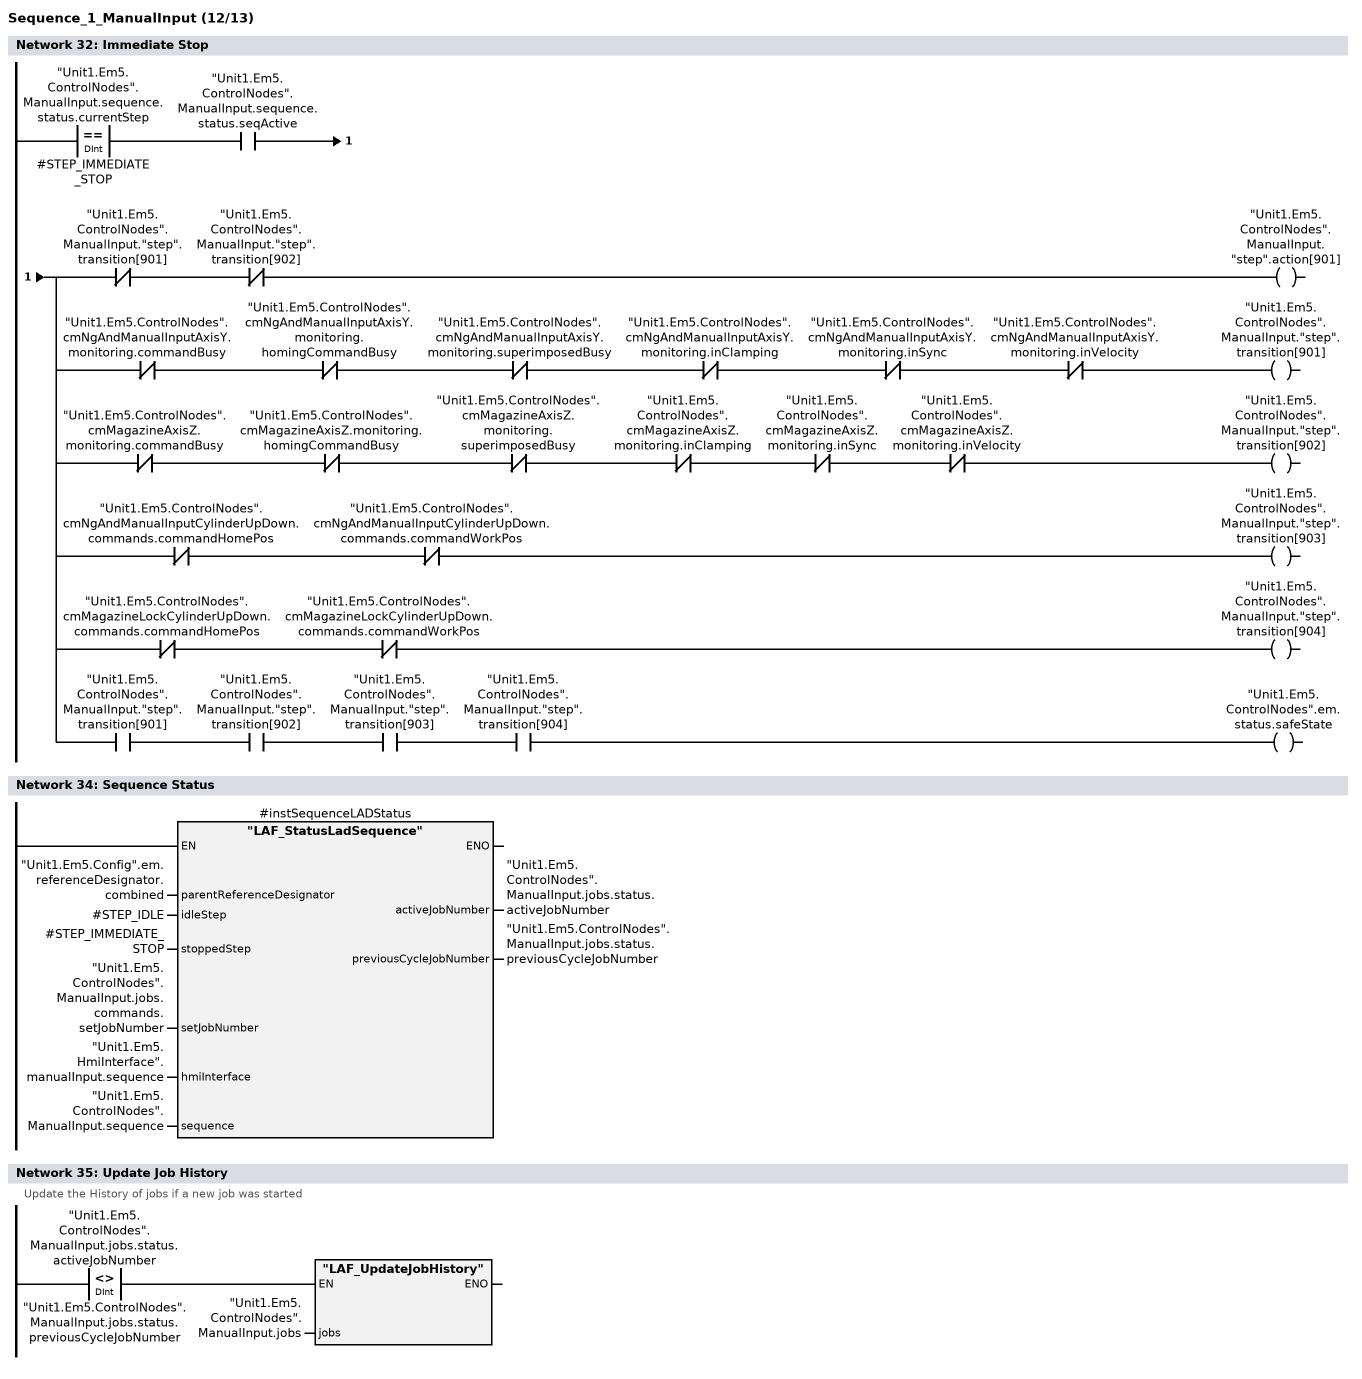
   RUNG wire#powerrail
      { S7_Templates := "SrcType := DInt" } EQ_Contact(in1 := "Unit1.Em5.ControlNodes".ManualInput.sequence.status.currentStep, in2 := #STEP_IMMEDIATE_STOP)
      Contact( "Unit1.Em5.ControlNodes".ManualInput.sequence.status.seqActive )
      wire#w1
      I_Contact( "Unit1.Em5.ControlNodes".ManualInput."step".transition[901] )
      I_Contact( "Unit1.Em5.ControlNodes".ManualInput."step".transition[902] )
      Coil( "Unit1.Em5.ControlNodes".ManualInput."step".action[901] )
   END_RUNG
   RUNG wire#w1
      I_Contact( "Unit1.Em5.ControlNodes".cmNgAndManualInputAxisY.monitoring.commandBusy )
      I_Contact( "Unit1.Em5.ControlNodes".cmNgAndManualInputAxisY.monitoring.homingCommandBusy )
      I_Contact( "Unit1.Em5.ControlNodes".cmNgAndManualInputAxisY.monitoring.superimposedBusy )
      I_Contact( "Unit1.Em5.ControlNodes".cmNgAndManualInputAxisY.monitoring.inClamping )
      I_Contact( "Unit1.Em5.ControlNodes".cmNgAndManualInputAxisY.monitoring.inSync )
      I_Contact( "Unit1.Em5.ControlNodes".cmNgAndManualInputAxisY.monitoring.inVelocity )
      Coil( "Unit1.Em5.ControlNodes".ManualInput."step".transition[901] )
   END_RUNG
   RUNG wire#w1
      I_Contact( "Unit1.Em5.ControlNodes".cmMagazineAxisZ.monitoring.commandBusy )
      I_Contact( "Unit1.Em5.ControlNodes".cmMagazineAxisZ.monitoring.homingCommandBusy )
      I_Contact( "Unit1.Em5.ControlNodes".cmMagazineAxisZ.monitoring.superimposedBusy )
      I_Contact( "Unit1.Em5.ControlNodes".cmMagazineAxisZ.monitoring.inClamping )
      I_Contact( "Unit1.Em5.ControlNodes".cmMagazineAxisZ.monitoring.inSync )
      I_Contact( "Unit1.Em5.ControlNodes".cmMagazineAxisZ.monitoring.inVelocity )
      Coil( "Unit1.Em5.ControlNodes".ManualInput."step".transition[902] )
   END_RUNG
   RUNG wire#w1
      I_Contact( "Unit1.Em5.ControlNodes".cmNgAndManualInputCylinderUpDown.commands.commandHomePos )
      I_Contact( "Unit1.Em5.ControlNodes".cmNgAndManualInputCylinderUpDown.commands.commandWorkPos )
      Coil( "Unit1.Em5.ControlNodes".ManualInput."step".transition[903] )
   END_RUNG
   RUNG wire#w1
      I_Contact( "Unit1.Em5.ControlNodes".cmMagazineLockCylinderUpDown.commands.commandHomePos )
      I_Contact( "Unit1.Em5.ControlNodes".cmMagazineLockCylinderUpDown.commands.commandWorkPos )
      Coil( "Unit1.Em5.ControlNodes".ManualInput."step".transition[904] )
   END_RUNG
   RUNG wire#w1
      Contact( "Unit1.Em5.ControlNodes".ManualInput."step".transition[901] )
      Contact( "Unit1.Em5.ControlNodes".ManualInput."step".transition[902] )
      Contact( "Unit1.Em5.ControlNodes".ManualInput."step".transition[903] )
      Contact( "Unit1.Em5.ControlNodes".ManualInput."step".transition[904] )
      Coil( "Unit1.Em5.ControlNodes".em.status.safeState )
   END_RUNG
   // the same network as SCL:
   #_w1 := ("Unit1.Em5.ControlNodes".ManualInput.sequence.status.currentStep = #STEP_IMMEDIATE_STOP) AND "Unit1.Em5.ControlNodes".ManualInput.sequence.status.seqActive;
   "Unit1.Em5.ControlNodes".ManualInput."step".action[901] := #_w1 AND NOT "Unit1.Em5.ControlNodes".ManualInput."step".transition[901] AND NOT "Unit1.Em5.ControlNodes".ManualInput."step".transition[902];
   "Unit1.Em5.ControlNodes".ManualInput."step".transition[901] := #_w1 AND NOT "Unit1.Em5.ControlNodes".cmNgAndManualInputAxisY.monitoring.commandBusy AND NOT "Unit1.Em5.ControlNodes".cmNgAndManualInputAxisY.monitoring.homingCommandBusy AND NOT "Unit1.Em5.ControlNodes".cmNgAndManualInputAxisY.monitoring.superimposedBusy AND NOT "Unit1.Em5.ControlNodes".cmNgAndManualInputAxisY.monitoring.inClamping AND NOT "Unit1.Em5.ControlNodes".cmNgAndManualInputAxisY.monitoring.inSync AND NOT "Unit1.Em5.ControlNodes".cmNgAndManualInputAxisY.monitoring.inVelocity;
   "Unit1.Em5.ControlNodes".ManualInput."step".transition[902] := #_w1 AND NOT "Unit1.Em5.ControlNodes".cmMagazineAxisZ.monitoring.commandBusy AND NOT "Unit1.Em5.ControlNodes".cmMagazineAxisZ.monitoring.homingCommandBusy AND NOT "Unit1.Em5.ControlNodes".cmMagazineAxisZ.monitoring.superimposedBusy AND NOT "Unit1.Em5.ControlNodes".cmMagazineAxisZ.monitoring.inClamping AND NOT "Unit1.Em5.ControlNodes".cmMagazineAxisZ.monitoring.inSync AND NOT "Unit1.Em5.ControlNodes".cmMagazineAxisZ.monitoring.inVelocity;
   "Unit1.Em5.ControlNodes".ManualInput."step".transition[903] := #_w1 AND NOT "Unit1.Em5.ControlNodes".cmNgAndManualInputCylinderUpDown.commands.commandHomePos AND NOT "Unit1.Em5.ControlNodes".cmNgAndManualInputCylinderUpDown.commands.commandWorkPos;
   "Unit1.Em5.ControlNodes".ManualInput."step".transition[904] := #_w1 AND NOT "Unit1.Em5.ControlNodes".cmMagazineLockCylinderUpDown.commands.commandHomePos AND NOT "Unit1.Em5.ControlNodes".cmMagazineLockCylinderUpDown.commands.commandWorkPos;
   "Unit1.Em5.ControlNodes".em.status.safeState := #_w1 AND "Unit1.Em5.ControlNodes".ManualInput."step".transition[901] AND "Unit1.Em5.ControlNodes".ManualInput."step".transition[902] AND "Unit1.Em5.ControlNodes".ManualInput."step".transition[903] AND "Unit1.Em5.ControlNodes".ManualInput."step".transition[904];
END_REGION

REGION Network 33: *************** STATUS **********************
END_REGION

REGION Network 34: Sequence Status
   RUNG wire#powerrail
      #instSequenceLADStatus(parentReferenceDesignator := "Unit1.Em5.Config".em.referenceDesignator.combined, idleStep := #STEP_IDLE, stoppedStep := #STEP_IMMEDIATE_STOP, setJobNumber := "Unit1.Em5.ControlNodes".ManualInput.jobs.commands.setJobNumber, hmiInterface := "Unit1.Em5.HmiInterface".manualInput.sequence, sequence := "Unit1.Em5.ControlNodes".ManualInput.sequence, activeJobNumber => "Unit1.Em5.ControlNodes".ManualInput.jobs.status.activeJobNumber, previousCycleJobNumber => "Unit1.Em5.ControlNodes".ManualInput.jobs.status.previousCycleJobNumber)
   END_RUNG
   // the same network as SCL:
   #instSequenceLADStatus(parentReferenceDesignator := "Unit1.Em5.Config".em.referenceDesignator.combined,   // "LAF_StatusLadSequence"
                          idleStep := #STEP_IDLE,
                          stoppedStep := #STEP_IMMEDIATE_STOP,
                          setJobNumber := "Unit1.Em5.ControlNodes".ManualInput.jobs.commands.setJobNumber,
                          hmiInterface := "Unit1.Em5.HmiInterface".manualInput.sequence,
                          sequence := "Unit1.Em5.ControlNodes".ManualInput.sequence,
                          activeJobNumber => "Unit1.Em5.ControlNodes".ManualInput.jobs.status.activeJobNumber,
                          previousCycleJobNumber => "Unit1.Em5.ControlNodes".ManualInput.jobs.status.previousCycleJobNumber);
END_REGION

REGION Network 35: Update Job History
   // Update the History of jobs if a new job was started
   RUNG wire#powerrail
      { S7_Templates := "SrcType := DInt" } NE_Contact(in1 := "Unit1.Em5.ControlNodes".ManualInput.jobs.status.activeJobNumber, in2 := "Unit1.Em5.ControlNodes".ManualInput.jobs.status.previousCycleJobNumber)
      "LAF_UpdateJobHistory"(jobs := "Unit1.Em5.ControlNodes".ManualInput.jobs)
   END_RUNG
   // the same network as SCL:
   IF "Unit1.Em5.ControlNodes".ManualInput.jobs.status.activeJobNumber <> "Unit1.Em5.ControlNodes".ManualInput.jobs.status.previousCycleJobNumber THEN
       "LAF_UpdateJobHistory"(jobs := "Unit1.Em5.ControlNodes".ManualInput.jobs);
   END_IF;
END_REGION

REGION Network 36: Output steps as String
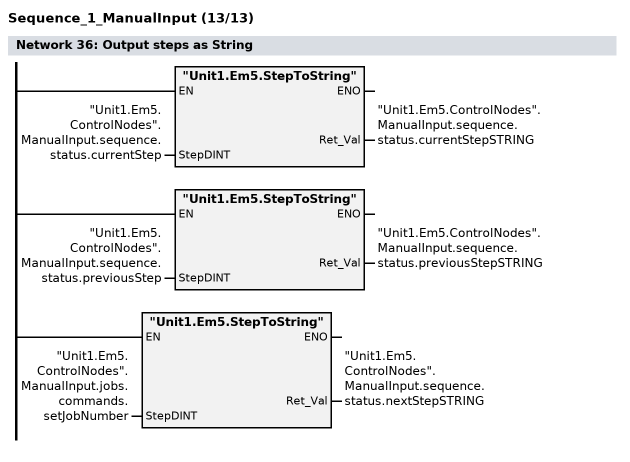
   RUNG wire#powerrail
      "Unit1.Em5.StepToString"(StepDINT := "Unit1.Em5.ControlNodes".ManualInput.sequence.status.currentStep, Ret_Val => "Unit1.Em5.ControlNodes".ManualInput.sequence.status.currentStepSTRING)
   END_RUNG
   RUNG wire#powerrail
      "Unit1.Em5.StepToString"(StepDINT := "Unit1.Em5.ControlNodes".ManualInput.sequence.status.previousStep, Ret_Val => "Unit1.Em5.ControlNodes".ManualInput.sequence.status.previousStepSTRING)
   END_RUNG
   RUNG wire#powerrail
      "Unit1.Em5.StepToString"(StepDINT := "Unit1.Em5.ControlNodes".ManualInput.jobs.commands.setJobNumber, Ret_Val => "Unit1.Em5.ControlNodes".ManualInput.sequence.status.nextStepSTRING)
   END_RUNG
   // the same network as SCL:
   "Unit1.Em5.ControlNodes".ManualInput.sequence.status.currentStepSTRING := "Unit1.Em5.StepToString"(StepDINT := "Unit1.Em5.ControlNodes".ManualInput.sequence.status.currentStep);
   "Unit1.Em5.ControlNodes".ManualInput.sequence.status.previousStepSTRING := "Unit1.Em5.StepToString"(StepDINT := "Unit1.Em5.ControlNodes".ManualInput.sequence.status.previousStep);
   "Unit1.Em5.ControlNodes".ManualInput.sequence.status.nextStepSTRING := "Unit1.Em5.StepToString"(StepDINT := "Unit1.Em5.ControlNodes".ManualInput.jobs.commands.setJobNumber);
END_REGION
END_FUNCTION_BLOCK
